(* CODESYS project tc3_cnc.library
   Company: Beckhoff Automation GmbH
   DefaultNamespace: Tc3_CNC
   Title: Tc3_CNC
   Description: TwinCAT CNC Library
   Placeholder: Tc3_CNC
   Author: Beckhoff Automation GmbH & Co. KG
   Version: 3.1.4000.18

Project tree, tasks and I/O mapping:
  libraries: Tc2_CncBase, * (Beckhoff Automation GmbH); Tc2_CncHli, * (Beckhoff Automation GmbH); Tc2_CncPlcopenP1, * (Beckhoff Automation GmbH); Tc2_EtherCAT, * (Beckhoff Automation GmbH); Tc2_Standard, * (Beckhoff Automation GmbH); Tc2_System, * (Beckhoff Automation GmbH); Tc2_Utilities, * (Beckhoff Automation GmbH); Tc3_Module, * (Beckhoff Automation GmbH)
  CNC/
    1 Init/
      program HLI3_Init [ST]
      function HLI3_SetAxisControlToPlc [ST]
      function HLI3_SetChannelControlToPlc [ST]
      function HLI3_UserInitialisation [ST]
    10 MessagesHandler/
      function CNCErrorDimensionToString [ST]
      function CNCErrorGetLogAxisId [ST]
      function CNCErrorMeaningToString [ST]
      function CNCErrorParameterToString [ST]
      function CNCErrorUnionToString [ST]
      function block FB_ChannelError [ST]
    11 Util/
      function F_GRAYCODE_TO_UINT [ST]
      function block FB_CNCWriteParameter [ST]
      function block FB_Uint_Udint [ST]
      function HLI3_FindAxisNameAndChannel [ST]
      function HLI3_FindHliAxisIdx [ST]
      function HLI3_GetEtherCATAxisInfo [ST]
      function block HLI3_SoftwareLimitSwitches [ST]
    12 CNC_Axis/
      function block FB_ActivateCompTable [ST]
      function block FB_CNCAxis [ST]
      function block FB_ReadSWLimitSwitches [ST]
      global variables GVL_CNC_AX
      function block HLI3_CNCAxis [ST]
      function block HLI3_CNCAxisBase [ST]: ACT_Init, ACT_Options, ACT_Parameter, ACT_PLCopen, ACT_Status
      data type ST_CNC_AX_Options
      data type ST_CNC_AX_Parameter
      data type ST_CNC_AX_PLCopen
      data type ST_CNC_AX_PLCopenStatus
      data type ST_CNC_AX_Status
    2 OperationMode/
      ModeManual/
        function HLI3_LogicalAxisInManualMode [ST]
        function block HLI3_ManualActivation [ST]
        function block HLI3_ManualExecution [ST]
        function block HLI3_ManualExecutionRapidMode [ST]
        function block HLI3_ManualModeHandler [ST]
        program PRG_AnalogJoystick [ST]
      function HLI3_AxisReset [ST]
      function HLI3_ChannelModeAuto [ST]
      function HLI3_ChannelModeManual [ST]
      function HLI3_ChannelModeMDI [ST]
      function HLI3_ChannelModeReference [ST]
      function HLI3_ChannelModeStandby [ST]
      function HLI3_ChannelReset [ST]
      function block HLI3_ChannelResetRequest [ST]
      function block HLI3_CNCChannel [ST]: AutoMDIStart, OpModes
      data type ST_CNC_CH_Options
    3 Control/
      function block FB_Diag [ST]
      function HLI3_ChannelSetBackwardMotion [ST]
      function HLI3_ChannelSetEmergencyStop [ST]
      function HLI3_ChannelSetFeedHold [ST]
      function HLI3_ChannelSetProgramBlockIgnore [ST]
      function HLI3_ChannelSetReducedFeed [ST]
      function HLI3_ChannelSetSingleBlock [ST]
      function HLI3_ChannelSetSuspendAxisOutput [ST]
      function HLI3_ClearReferencePosition [ST]
      function HLI3_GetActualAxisPos [ST]
      function HLI3_GetAxisReferenceState [ST]
      function block HLI3_GetChannelActiveG [ST]
      function HLI3_GetChannelError [ST]
      function block HLI3_GetChannelMessage [ST]
      function HLI3_GetChannelMode [ST]
      function HLI3_GetChannelState [ST]
      function HLI3_GetChannelStatusInfo [ST]
      function HLI3_GetFeedholdState [ST]
      function HLI3_GetIpoState [ST]
      function block HLI3_HandleSpindleTechno [ST]: A_HandleTechno, M_HandleTechnoAx, M_HandleTechnoCh, M_ManageAcknowledgement
      function block HLI3_HandleSpindleTechnoGearchange [ST]
      function HLI3_SetAxisGantryOn [ST]
      function HLI3_SetAxisOverride [ST]
      function HLI3_SetAxisReferenceCam [ST]
      function block HLI3_SetAxisReferenceOffset [ST]
      function HLI3_SetAxisReferencePosition [ST]
      function block HLI3_SetAxisRelease [ST]: AC_CanOpenDrive, AC_ClearError, AC_SercosDrive, AC_TerminalDrive
      function block HLI3_SetAxisSpindleStopAtProgramEnd [ST]
      function HLI3_SetAxisTrackingOperation [ST]
      function HLI3_SetChannelOverride [ST]
      function HLI3_SetChannelRapidOverride [ST]
      function HLI3_SetProbingSignal [ST]
    4 MHT-Function/
      function HLI3_ChannelResetHFunctions [ST]
      function HLI3_ChannelResetMFunctions [ST]
      function block HLI3_DoChannelHFunction [ST]
      function block HLI3_DoChannelMFunction [ST]
      function block HLI3_DoChannelTFunction [ST]
      function block HLI3_FastMFunctionHandler [ST]: ClearQueue, Dequeue, DequeuingRequired, Enqueue, RefreshQueue
      function block HLI3_FastMFunctionProvider [ST]
      function HLI3_QuitAxisMFunction [ST]
      function block HLI3_QuitChannelMHTFunction [ST]
    5 Variables/
      function block FB_ReadCNCVariables [ST]
      function HLI3_GetVEChannelBooleanValue [ST]
      function HLI3_GetVEChannelDIntValue [ST]
      function HLI3_GetVEChannelLRealValue [ST]
      function HLI3_GetVEChannelStringValue [ST]
      function HLI3_LinkVEChannelStructure [ST]
      function HLI3_SetVEChannelBooleanValue [ST]
      function HLI3_SetVEChannelDIntValue [ST]
      function HLI3_SetVEChannelLRealValue [ST]
      function HLI3_SetVEChannelStringValue [ST]
    6 BlockSearch/
      function block HLI3_BlockSearch [ST]
      function block ReadBlockCount [ST]
      function block ReadBlockNumber [ST]
      function block ReadBsAutoReturn [ST]
      function block ReadBsBlockCount [ST]
      function block ReadBsBlockNumber [ST]
      function block ReadBsCoveredDistance [ST]
      function block ReadBsDeviationMax [ST]
      function block ReadBsPass [ST]
      function block ReadBsType [ST]
      function block WriteBsAutoReturn [ST]
      function block WriteBsBlockCount [ST]
      function block WriteBsBlockNumber [ST]
      function block WriteBsCoveredDistance [ST]
      function block WriteBsDeviationMax [ST]
      function block WriteBsPass [ST]
      function block WriteBsType [ST]
    7 ToolManagement/
      program HLI3_ToolManagement [ST]: D_Command, T_Command, ToolLife_Command
    8 Mis/
      function block FB_WriteCNCZeroOffset [ST]
      function block FB_WriteCNCZeroOffsetDefault [ST]
      function block HLI_HandleMessages [ST]
      function block HLI_MoveSpindle [ST]
      function HLI3_CheckAxisValid [ST]
      function HLI3_CheckChannelValid [ST]
      program HLI3_CheckCNCAlive [ST]
      function HLI3_GetHliAxisIdx [ST]
      function HLI3_GetHliChannelIdx [ST]
      function HLI3_GetLogAxisId [ST]
      function HLI3_ResetSpindle [ST]
      function HLI3_SetPLCAlive [ST]
      program PB_10_CNC_Spindelkopplung [ST]
  DUTs/
    CNC_DataTyps/
      data type E_HLI_MM_KEYDIRECTION
      interface ITF_ToolAction: Commit, Tool
      data type ST_BlockSearch
      data type ST_ChannelSignals
      data type ST_CNC_TOOL_DATA_EXT
      data type ST_CNC_ToolChannel
      data type ST_CNCAxis
      data type ST_CncChannel
      data type ST_CncChannelInfo
      data type ST_CNCCmdModesStates
      data type ST_CNCG159VG
      data type ST_CncSystem
      data type ST_ManualMode
      data type ST_OpModes
      data type ST_OpStates
      data type ST_SyntaxCheck
      data type ST_TechnoAttributeData
      data type VEData
    CNC_FastMFunction/
      data type E_FastMFunctionState
      data type ST_FastMFunctionBufferItem
      data type ST_FastMFunctionData
      data type ST_FastMFunctionItem
    CNC_ManualMode/
      data type E_CNC_ManualType
      data type E_CNC_ManualZeroOffset
      data type ST_CNC_ManualOption
      data type ST_ManualModeAxis
      data type ST_ManualModeAxisKeys
      data type ST_ManualModeAxisParameter
      data type ST_ManualModeChannelParameter
      data type ST_ManualModeControlElements
      data type ST_ManualModeControlElementState
      data type ST_ManualModeJoystickParameter
      data type ST_ManualModeKeyHWUnit
      data type ST_ManualModeParameter
      data type ST_ManualModeState
    CNC_VariablesViewer/
      data type E_CNCVariablesType
      data type E_VEVariablesType
      data type ST_CNCVariablesViewer_Data
    CNC_WriteParameter/
      data type E_CNCParameterTypes
      data type ST_CNCParameter
    EventLogger/
      data type E_LogMethod
      data type ST_EventData
      data type ST_FileInfo
  GVLs/
    global variables Global_CNC
    global variables Global_CNCVariablesViewer
    global variables Global_ManualMode
  Version/
    global variables Global_Version
  Tc3_CNC.tmc
*)

// CNC/12 CNC_Axis/ST_CNC_AX_Options
TYPE ST_CNC_AX_Options :
STRUCT
	bResetCalibration	: BOOL;
	bReducedSpeed 		: BOOL;
	bReducedSpeedZone1  : BOOL;
	bReducedSpeedZone2  : BOOL;
	bProbingSignal		: BOOL;
	bActivateCompTable	: BOOL;	 
	strPathCompTable	: STRING(256);
END_STRUCT
END_TYPE

// CNC/12 CNC_Axis/ST_CNC_AX_Parameter
TYPE ST_CNC_AX_Parameter :
STRUCT
	nNumParameters 		: INT; 	
	bWriteParameter     : BOOL;	
	strTempPath			: STRING;
	ParamList			: ARRAY[0..199] OF ST_CNCParameter;
END_STRUCT
END_TYPE

// CNC/12 CNC_Axis/ST_CNC_AX_PLCopen
TYPE ST_CNC_AX_PLCopen :
STRUCT	
	nOverride 		     : UINT; 		// [ 0.1% ]
	bExecuteHoming		 : BOOL;
	bCamSignal			 : BOOL;
	bExecuteMoveAbsolute : BOOL;
 	bExecuteStop 		 : BOOL;
	bExecuteReset 		 : BOOL;	
	fPosition 			 : LREAL;      // [ mm or degree ]
	fVelocity       	 : LREAL;      // [ mm/min or degree/min ]
	fAcceleration   	 : LREAL;	  // [ mm/s^2 or degree/s^2 ]
	fJerk   			 : LREAL;	  // [ mm/s^3 or degree/s^3 ]
END_STRUCT
END_TYPE

// CNC/12 CNC_Axis/ST_CNC_AX_PLCopenStatus
TYPE ST_CNC_AX_PLCopenStatus :
STRUCT	
	bError 				: BOOL;
	nErrorID 			: DINT;
	bMoveAbsoluteDone 	: BOOL;
	bHomingDone 		: BOOL;
	bStopDone 			: BOOL;
	bResetDone 			: BOOL;
END_STRUCT
END_TYPE

// CNC/12 CNC_Axis/ST_CNC_AX_Status
TYPE ST_CNC_AX_Status :
STRUCT
	bHomingDone 	: BOOL;
	fSetPosACS		: LREAL;	// [ mm or degree ] 
	fActPosACS		: LREAL;	// [ mm or degree] 
	fActVelo		: LREAL;	// [ mm or degree or rpm ]
	nCNCErrorID 	: UDINT;	// CNC Axis Error Id
	PLCopen   		: ST_CNC_AX_PLCopenStatus;
END_STRUCT
END_TYPE

// CNC/2 OperationMode/ST_CNC_CH_Options
TYPE ST_CNC_CH_Options :
STRUCT
	bReferenceModeStartRequired : BOOL;
END_STRUCT
END_TYPE

// DUTs/CNC_DataTyps/E_HLI_MM_KEYDIRECTION
TYPE E_HLI_MM_KEYDIRECTION :
(
	KEY_DIR_NEGATIVE := -1,
	KEY_DIR_NOT_PRESSED := 0,
	KEY_DIR_POSITIVE := 1
);
END_TYPE

// DUTs/CNC_DataTyps/ST_BlockSearch
TYPE ST_BlockSearch :
STRUCT
	/// Block Search 
	Active: BOOL;
	/// Edge signal 
	bStartRead: BOOL;
	/// Edge signal 
	bStartWrite: BOOL;
	/// 0 - no block search
	///                                    3 - start position by block count
	///                                    4 - start position by block nr
	///                                    5 - start position BY individual mark 
	nType: UINT;
	fDistance: LREAL;
	bAutoReturn: BOOL;
	nDeviationMax: UDINT;
	nBlockNumber: DINT;
	nPass: DINT;
	nBlockCount: DINT;
END_STRUCT
END_TYPE

// DUTs/CNC_DataTyps/ST_ChannelSignals
TYPE ST_ChannelSignals :
STRUCT
	DoSingleBlock: BOOL;
	SingleBlock: BOOL;
	FeedHold: BOOL;
	Backward: BOOL;
	PrgBlockIgnore: BOOL;
	M01Stop: BOOL;
END_STRUCT
END_TYPE

// DUTs/CNC_DataTyps/ST_CNC_TOOL_DATA_EXT
TYPE ST_CNC_TOOL_DATA_EXT :
STRUCT
	tool_desc: CNC_TOOL_DESC;
	tool_life: CNC_TOOL_LIFE_DATA;
	dist_max: LREAL;
	time_max: LREAL;
	/// 0.1 µm 
	laenge: DINT;
	/// 0.1 µm 
	laenge_delta: DINT;
	/// 0.1 µm 
	radius: DINT;
	/// 0.1 µm 
	radius_delta: DINT;
	/// position in tool holder 
	pos: DINT;
	/// 0.1 µm 
	tolerancePos: DINT;
	/// 0.1 µm 
	toleranceNeg: DINT;
END_STRUCT
END_TYPE

// DUTs/CNC_DataTyps/ST_CNC_ToolChannel
TYPE ST_CNC_ToolChannel :
STRUCT
	
	bToolRequest: 			BOOL;   (* rising edge starts request of tool data from HMI, HMI resets to false after reading *)
	nToolRequestID: 		DINT;   (* tool id for request *)
	nToolRequestIDSister:	DINT;	(* tool sister id for request, 0 if not needed *)
	nToolRequestIDVariant:	DINT;   (* tool variant id for request, 0 if not needed *)		
	
	bToolRequestPrepData:	BOOL;   (* rising edge starts request of tool data to structure stPrepTool *)
	nToolRequestPrepId: 	DINT;   (* tool id for pepRequest *)
	
	bOldToolDataExist:		BOOL;   (* rising edge commands the HMI to read oldData from stOldTool *)
		
	stActTool:	 			ST_CNC_TOOL_DATA_EXT; (* complete tool data for actual tool that will be transfered FROM HMI  *)
	stOldTool:	 			ST_CNC_TOOL_DATA_EXT; (* complete tool data for odlTool that will be transfered TO HMI *)
	stPrepTool:				ST_CNC_TOOL_DATA_EXT; (* complete tool data for preTool that will be transfered FROM HMI *)
	
	stActT:					ST_CNC_TOOL_DATA_EXT; (* (internal) tool data for the actual requested T *)
	
	nToolInCnc:				DINT;	(* main tool id of tool actually in cnc *)
	nToolInCncSister: 		DINT;	(* sister tool id of tool actually in cnc *)
	nToolInCncVariant:		DINT;	(* variant tool id of tool actually in cnc *)
	
	bResetToolRequest:		BOOL;
	
	TCommand:				ITF_ToolAction;  (* the method Commit is called before data for T is transfered to CNC. The process os stopped until the commit method returns true *)
	DCommand:				ITF_ToolAction;  (* the method Commit is called before data for D is transfered to CNC. The process os stopped until the commit method returns true *)
	ToolLifeCommand:		ITF_ToolAction;  (* the method Commit is called before data for ToolLife is transfered to HMI. The process os stopped until the commit method returns true *)	

END_STRUCT
END_TYPE

// DUTs/CNC_DataTyps/ST_CNCAxis
TYPE ST_CNCAxis :
STRUCT
	nHliAxisIdx : INT := -1;
    strLogName	: STRING(HLI_ACHS_NAME_LAENGE);
	{attribute 'hide'}
	nCNCErrorID : UDINT;	
END_STRUCT
END_TYPE

// DUTs/CNC_DataTyps/ST_CncChannel
TYPE ST_CncChannel :
STRUCT
	nLogNumber  : DINT := -1;
    strLogName	: STRING(HLI_ACHS_NAME_LAENGE);
	/// Operation Mode 
	Mode: ST_OpModes;
	/// Operation States 
	State: ST_OpStates;
	/// Selected Mode 
	ActMode: UDINT;
	/// Selected Mode as string 
	ActModeString: STRING;
	/// Selected State 
	ActState: UDINT;
	/// Selected State as string 
	ActStateString: STRING;
	/// Block Search : Act. Distance 
	ActDistance: LREAL;
	/// Block Search : Act. Block Count 
	ActBlockCount: UDINT;
	actM_r: STRING(5);
	actH_r: STRING(5);
	/// M-Functions 
	M: ARRAY[0..999] OF ST_TechnoAttributeData;
	/// H-Functions 
	H: ARRAY[0..999] OF ST_TechnoAttributeData;	
	/// Fehlerflag des Kanals 
	Error: BOOL;	
	/// Message from NC program to PLC 
	Message: STRING(HLI_MSG_CONTENT_STRL);
	// Data for tool handling
	ToolData      :  ST_CNC_ToolChannel;
	
END_STRUCT
END_TYPE

// DUTs/CNC_DataTyps/ST_CncChannelInfo
TYPE ST_CncChannelInfo :
STRUCT
	nHliChannelIdx : INT := -1;
    strLogName	: STRING(HLI_CHANNEL_NAME_LAENGE);
END_STRUCT
END_TYPE

// DUTs/CNC_DataTyps/ST_CNCCmdModesStates
TYPE ST_CNCCmdModesStates :
	STRUCT	
	stModes : ST_OpModes;
	stStates : ST_OpStates;
	END_STRUCT
END_TYPE

// DUTs/CNC_DataTyps/ST_CNCG159VG
TYPE ST_CNCG159VG :
STRUCT
	sTarget: STRING(95);
	dValue: DINT;
END_STRUCT
END_TYPE

// DUTs/CNC_DataTyps/ST_CncSystem
TYPE ST_CncSystem :
STRUCT
	/// Initialization of HLI done 
	bHLIInit: BOOL;
	/// Initialization of PLCopenPlatform done 
	bPLCopenPlatformInit : BOOL;
	/// Initialization of user data done
	bUserInitDone: BOOL;
	/// Error init HLI-Interfaces 
	bInitError: BOOL;
	/// ErrorId during init HLI-Interfaces 
	nInitErrorId: UDINT;
	Channel: ARRAY[0..HLI_SYS_CH_MAXIDX] OF ST_CncChannel;
    LogAxisNo : ARRAY[0..MAX_SYS_LOG_AXIS_INDEX] OF ST_CncAxis;	
	LogChannelNo : ARRAY[0..HLI_SYS_CH_MAXIDX] OF ST_CncChannelInfo;    	
END_STRUCT
END_TYPE

// DUTs/CNC_DataTyps/ST_ManualMode
TYPE ST_ManualMode :
STRUCT
	bKeyPos: BOOL;
	bKeyNeg: BOOL;
	bKeyRapid: BOOL;
	nLogAxisNumber: UINT;
	nInc: UDINT;
	nManualTyp: UINT;
	stManualOption			: ST_CNC_ManualOption;
	nSpeed: UINT;
	/// Handradauflösung in 0.1 um / Umdrehung 
	nHwResolution: UDINT;
END_STRUCT
END_TYPE

// DUTs/CNC_DataTyps/ST_OpModes
TYPE ST_OpModes :
STRUCT
	Standby: BOOL;
	Auto: BOOL;
	Manual: BOOL;
	MDI: BOOL;	
	Homing: BOOL;
END_STRUCT
END_TYPE

// DUTs/CNC_DataTyps/ST_OpStates
TYPE ST_OpStates :
STRUCT
	Selected: BOOL;
	Ready: BOOL;
	Active: BOOL;
	Hold: BOOL;
	Reset: BOOL;
END_STRUCT
END_TYPE

// DUTs/CNC_DataTyps/ST_SyntaxCheck
TYPE ST_SyntaxCheck :
STRUCT
	/// SyntaxCheck 
	nType: INT;
END_STRUCT
END_TYPE

// DUTs/CNC_DataTyps/ST_TechnoAttributeData
TYPE ST_TechnoAttributeData :
STRUCT
	bState_rw: BOOL;
	nFunctionNumber_r: UDINT;
	nTime_r: DINT;
	nBlockNumber_r: UDINT;
	nPrgLineNumber_r: UDINT;
	nArgument_r: DINT;
	{attribute 'hide'}
	bRes: BOOL;
END_STRUCT
END_TYPE

// DUTs/CNC_DataTyps/VEData
TYPE VEData :
STRUCT
	AHLI_UNS32_Data: ARRAY[0..HLI_EXT_VAR32_MAXIDX] OF UDINT;
END_STRUCT
END_TYPE

// DUTs/CNC_FastMFunction/E_FastMFunctionState
(****************************************************************************************)
(* POU:		E_FastMFunctionState                     									*)
(* Type:	ENUM																		*)
(* Author: 	RCH		                                             						*)
(* Date: 	14/10/29																	*)
(* Rev.: 	1.0                                               							*)
(* ------------------------------------------------------------------------------------ *)
(* Desc.:	Defines the state of an digital output handled by instances of FB			*)
(*			HLI3_FastMFunctionHandler.													*)
(* ------------------------------------------------------------------------------------ *)
(* Rev.:	<Enter revision number here>												*)
(* Date:	<Enter revision data here>				                                   	*)
(* Author:	<Enter author´s shortcut here>											 	*)
(* Desc.:	<Enter description here>													*)
(****************************************************************************************)
TYPE E_FastMFunctionState :
(
	EMPTY	:= 0,	(* Not switched yet *)
	OFF 	:= 1,	(* Switched OFF *)
	ON 		:= 2	(* Switched ON *)
);
END_TYPE

// DUTs/CNC_FastMFunction/ST_FastMFunctionBufferItem
(****************************************************************************************)
(* POU:		ST_FastMFunctionBufferItem                     								*)
(* Type:	STRUCT																		*)
(* Author: 	RCH		                                             						*)
(* Date: 	14/10/29																	*)
(* Rev.: 	1.0                                               							*)
(* ------------------------------------------------------------------------------------ *)
(* Desc.:	Defines data content for a single fast M function switch event managed 		*)
(*			internally by instances of HLI3_FastMFunctionHandler.						*) 
(* ------------------------------------------------------------------------------------ *)
(* Rev.:	<Enter revision number here>												*)
(* Date:	<Enter revision data here>				                                   	*)
(* Author:	<Enter author´s shortcut here>											 	*)
(* Desc.:	<Enter description here>													*)
(****************************************************************************************)
TYPE ST_FastMFunctionBufferItem :
STRUCT
	eState			: E_FastMFunctionState;		(* The target switch state *)
	nSwitchTime		: DINT;						(* The calculated switch time *)
END_STRUCT
END_TYPE

// DUTs/CNC_FastMFunction/ST_FastMFunctionData
(****************************************************************************************)
(* POU:		ST_FastMFunctionData                     								*)
(* Type:	STRUCT																		*)
(* Author: 	RCH		                                             						*)
(* Date: 	14/10/29																	*)
(* Rev.: 	1.0                                               							*)
(* ------------------------------------------------------------------------------------ *)
(* Desc.:	Defines preprocessed information about MOS_TS M functions and their			*)
(*			metadata generated by HLI3_FastMFunctionProvider and consumed by 			*)
(*			HLI3_FastMFunctionHandler(s)												*) 
(* ------------------------------------------------------------------------------------ *)
(* Rev.:	<Enter revision number here>												*)
(* Date:	<Enter revision data here>				                                   	*)
(* Author:	<Enter author´s shortcut here>											 	*)
(* Desc.:	<Enter description here>													*)
(****************************************************************************************)
TYPE ST_FastMFunctionData :
STRUCT
	bCycleTimeExceeded	: BOOL;																	(* TRUE if the cycle time has been exceeded and therefore the data is unvalid *)
	bDataValid			: BOOL;																	(* TRUE if data is valid *)
	nFunctionCount		: UINT;																	(* Number of M function data sets contained in 'astItem' *)
	astItem				: ARRAY[0..MAX_FAST_M_FUNC_ITEM_IDX] OF ST_FastMFunctionItem;			(* M function metadata items *)
END_STRUCT
END_TYPE

// DUTs/CNC_FastMFunction/ST_FastMFunctionItem
(****************************************************************************************)
(* POU:		ST_FastMFunctionItem                     									*)
(* Type:	STRUCT																		*)
(* Author: 	RCH		                                             						*)
(* Date: 	14/10/29																	*)
(* Rev.: 	1.0                                               							*)
(* ------------------------------------------------------------------------------------ *)
(* Desc.:	Defines M function metadata content provided by HLI3_FastMFunctionProvider	*)
(* ------------------------------------------------------------------------------------ *)
(* Rev.:	<Enter revision number here>												*)
(* Date:	<Enter revision data here>				                                   	*)
(* Author:	<Enter author´s shortcut here>											 	*)
(* Desc.:	<Enter description here>													*)
(****************************************************************************************)
TYPE ST_FastMFunctionItem :
STRUCT
	nFunctionNo		: UINT;			(* M function number *)
	nOffset			: DINT;			(* Time offset with respect to the block change time *)
	nCycleCount		: UDINT;		(* PLC cycle counter *)
END_STRUCT
END_TYPE

// DUTs/CNC_ManualMode/E_CNC_ManualType
TYPE E_CNC_ManualType :
(
	NoManualMode := 0,
	Handwheel := 1,
	TippMode := 2,
	JogMode := 3,
	JoystickMode := 4,
	DigitalJoystick := 5
);
END_TYPE

// DUTs/CNC_ManualMode/E_CNC_ManualZeroOffset
TYPE E_CNC_ManualZeroOffset :
(
	G53 := 0,
	G54 := 1,
	G55 := 2,
	G56 := 3,
	G57 := 4,
	G58 := 5,
	G59 := 6
);
END_TYPE

// DUTs/CNC_ManualMode/ST_CNC_ManualOption
TYPE ST_CNC_ManualOption :
STRUCT
	bTrafoActive: BOOL;
	bEcsActive: BOOL;
	bCAXActive: BOOL;
	eZeroOffset: E_CNC_ManualZeroOffset;
END_STRUCT
END_TYPE

// DUTs/CNC_ManualMode/ST_ManualModeAxis
TYPE ST_ManualModeAxis :
STRUCT
	nLogAxisNr: UINT;
	nSpeed: UDINT;
END_STRUCT
END_TYPE

// DUTs/CNC_ManualMode/ST_ManualModeAxisKeys
TYPE ST_ManualModeAxisKeys :
STRUCT
	/// static signal + 
	bKeyPos: BOOL;
	/// static signal - 
	bKeyNeg: BOOL;
	/// static signal Rapid 
	bKeyRapid: BOOL;
END_STRUCT
END_TYPE

// DUTs/CNC_ManualMode/ST_ManualModeAxisParameter
TYPE ST_ManualModeAxisParameter :
STRUCT
	stControlUnit: ARRAY[0..HLI_KEY_MAXIDX] OF ST_ManualModeAxis;
END_STRUCT
END_TYPE

// DUTs/CNC_ManualMode/ST_ManualModeChannelParameter
TYPE ST_ManualModeChannelParameter :
STRUCT
	/// Number of channel 
	nChanIdx: INT := -1;
	nInc: UDINT;
	/// Aufloesung des Achsverfahrwegs bei einer Handradumdrehung Einheit: 0.1um / Handradumdrehung
	nHandwheelResolution: DINT;	 	
	/// configuration 
	eManualType: E_CNC_ManualType;
	stManualOption: ST_CNC_ManualOption;
	strInitParameter: STRING;
END_STRUCT
END_TYPE

// DUTs/CNC_ManualMode/ST_ManualModeControlElements
TYPE ST_ManualModeControlElements :
STRUCT
	stControlKeys: ARRAY[0..HLI_KEY_MAXIDX] OF ST_ManualModeAxisKeys;
	stControlJoystickValue: ARRAY[0..HLI_KEY_MAXIDX] OF DINT;
	/// Es können 6 Handräder verwendet werden 
	nHandwheelInc: ARRAY[0..HLI_HW_MAXIDX] OF DINT;
END_STRUCT
END_TYPE

// DUTs/CNC_ManualMode/ST_ManualModeControlElementState
TYPE ST_ManualModeControlElementState :
STRUCT
	stKeyUnit: ARRAY[0..HLI_KEY_MAXIDX] OF ST_ManualModeKeyHWUnit;
	stHWUnit: ARRAY[0..HLI_HW_MAXIDX] OF ST_ManualModeKeyHWUnit;
END_STRUCT
END_TYPE

// DUTs/CNC_ManualMode/ST_ManualModeJoystickParameter
TYPE ST_ManualModeJoystickParameter :
STRUCT
	/// static signal : Analog Min Value 
	AnalogValueMin: DINT;
	/// static signal : Analog Max Value 
	AnalogValueMax: DINT;
	/// Dead Band for Zero Value 
	AnalogValueZeroDeadBand: DINT;
END_STRUCT
END_TYPE

// DUTs/CNC_ManualMode/ST_ManualModeKeyHWUnit
TYPE ST_ManualModeKeyHWUnit :
STRUCT
	nLogAxisId: UINT;
	nChan: INT := -1;
	nInputParameterIdx: INT;
END_STRUCT
END_TYPE

// DUTs/CNC_ManualMode/ST_ManualModeParameter
TYPE ST_ManualModeParameter :
STRUCT
	stAxisParameter: ST_ManualModeAxisParameter;
	stJoystickParameter: ST_ManualModeJoystickParameter;
	stChannelParameter: ST_ManualModeChannelParameter;	
END_STRUCT
END_TYPE

// DUTs/CNC_ManualMode/ST_ManualModeState
TYPE ST_ManualModeState :
STRUCT
	arrAxisInG201: ARRAY[0..HLI_KEY_MAXIDX] OF UINT;
END_STRUCT
END_TYPE

// DUTs/CNC_VariablesViewer/E_CNCVariablesType
{attribute 'qualified_only'}
{attribute 'strict'}
TYPE E_CNCVariablesType :
(
	none :=0,
	VE,
    P,
    VP,
    VS,
    VL        
);
END_TYPE

// DUTs/CNC_VariablesViewer/E_VEVariablesType
{attribute 'qualified_only'}
{attribute 'strict'}
TYPE E_VEVariablesType :
(
	none := 0,
	BOOLEAN,
	SGN08,
	UNS08,
	SGN16,
	UNS16,
	SGN32,
	UNS32,
	REAL64,
	VESTRING	
);
END_TYPE

// DUTs/CNC_VariablesViewer/ST_CNCVariablesViewer_Data
TYPE ST_CNCVariablesViewer_Data :
STRUCT
	strName : STRING;
	strValue  : STRING(799);
END_STRUCT
END_TYPE

// DUTs/CNC_WriteParameter/E_CNCParameterTypes
TYPE E_CNCParameterTypes :
(
	CNC_ChannelParameter := 10,
	CNC_AxisParameter := 11,
	CNC_ZeroOffsets := 12,
	CNC_ToolParameter := 13,
	CNC_ClampPosition := 14
);
END_TYPE

// DUTs/CNC_WriteParameter/ST_CNCParameter
TYPE ST_CNCParameter :
STRUCT
	strName: STRING;
	strValue: STRING;
	strDescription: STRING;
END_STRUCT
END_TYPE

// DUTs/EventLogger/E_LogMethod
TYPE E_LogMethod :
(
	Static := 0,
	RisingTrig := 1,
	FallingTrig := 2
);
END_TYPE

// DUTs/EventLogger/ST_EventData
TYPE ST_EventData :
STRUCT
	nParam1: DINT;
	nParam2: STRING;	
END_STRUCT
END_TYPE

// DUTs/EventLogger/ST_FileInfo
TYPE ST_FileInfo :
STRUCT
	nSource: UDINT;
	nOffset: UDINT;
	sFilename: STRING(260);
END_STRUCT
END_TYPE

// CNC/12 CNC_Axis/GVL_CNC_AX
VAR_GLOBAL
	fbCNC_AX_WriteParameter			: FB_CNCWriteParameter;	
	bCNC_AX_WriteParameterLock 		: BOOL;
	fbActivateCompTable 			: FB_ActivateCompTable;
	bCNC_AX_ActivateCompTableLock  	: BOOL;
END_VAR

// GVLs/Global_CNC
VAR_GLOBAL
	CNCSystem						: ST_CncSystem;
END_VAR

(****************************************************************************************)
(*	  	Global constants used by the fast M function handling process (MOS_TS)			*)
(****************************************************************************************)
VAR_GLOBAL CONSTANT
	MAX_FAST_M_FUNC_ITEM_IDX	: UINT	:= 7;			(* Max. index of fast M functions processed by HLI3_FastMFunctionProvider per PLC cycle *) 
	MAX_FAST_M_FUNC_QUEUE_IDX	: UINT	:= 63;			(* Max. index of fast M function switch events buffered by HLI3_FastMFunctionHandler *) 
	MAX_FAST_M_FUNC_OUTPUT_IDX	: UINT	:= 124;			(* Max. index of fast M function oversampling output byte array *)			
	MAX_SYS_LOG_AXIS_INDEX		: UINT  := 255;			(* Max. Index of Log. Axis Id *) 				
END_VAR

// GVLs/Global_CNCVariablesViewer
{attribute 'pack_mode' := '1'}
VAR_GLOBAL
	stCNCVariablesViewer_Data : ARRAY[0..MAX_CNC_VAR_LIST_IDX] OF ST_CNCVariablesViewer_Data;
	eVariablesType : E_CNCVariablesType;

END_VAR

VAR_GLOBAL CONSTANT
	MAX_CNC_VAR_LIST_IDX : UINT := 200;
END_VAR

// GVLs/Global_ManualMode
VAR_GLOBAL
	/// Manual mode control structures 
	stManualModeParameter: ARRAY[0..HLI_SYS_CH_MAXIDX] OF ST_ManualModeParameter;
	stManualModeControlElements: ARRAY[0..HLI_SYS_CH_MAXIDX] OF ST_ManualModeControlElements;
	stManualModeState: ARRAY[0..HLI_SYS_CH_MAXIDX] OF ST_ManualModeState;
	stManualModeControlElementState : ST_ManualModeControlElementState;
END_VAR

// Version/Global_Version
{attribute 'TcGenerated'}
// This function has been automatically generated from the project information.
VAR_GLOBAL CONSTANT
	{attribute 'const_non_replaced'}
	{attribute 'linkalways'}
	stLibVersion_Tc3_CNC : ST_LibVersion := (iMajor := 3, iMinor := 1, iBuild := 4000, iRevision := 18, sVersion := '3.1.4000.18');
END_VAR

// CNC/1 Init/HLI3_Init
PROGRAM HLI3_Init
VAR
	Hli: MCV_HliInterface;
	bFirstCycle: BOOL := TRUE;
	ipSrv: ITComObjectServer;
	oidCnc: UDINT := 16#5500001;
	bUnregister: BOOL;
	MessageOutput: R_TRIG;
	nHliAxisIdx	: INT;
	nHliChannelIdx: INT;
	
	PlatformBase: MCV_PlatformBase;
	P1_Platform: MCV_P1_Platform;
END_VAR

(* ========================================================= *)
(*    PRG: HLI_Init                                          *)
(* --------------------------------------------------------- *)
(*   Desc:                                                   *)
(* Author: MK                                                *)
(*   Date: 21.12.2011                                        *)
(*   Rev.: 1.0                                               *)
(*   Date: 06.08.2013                                        *)
(*   Rev.: 1.1 TV   Error Message if HLI not initialized	 *)
(*   Date: 05.01.2017                                        *)
(*   Rev.: 1.2 TV   BugFix Init LogAxisNo Array              *)
(*   Date: 06.06.2017                                        *)
(*   Rev.: 1.3 TV  new LogChannelNo            	 			 *)
(*   Date: 08.11.2017                                        *)
(*   Rev.: 1.4 TV  new FB call fbCNC_AX_WriteParameter       *)
(*   			   new FB call 	fbActivateCompTable       	 *)
(* ========================================================= *)



IF bFirstCycle THEN
	Hli();					(* initialize HLI *)
	bFirstCycle := FALSE;
END_IF


IF Hli.Initialized  = TRUE
THEN
	(* User initialization, used during start of PLC once *)
	IF CncSystem.bUserInitDone = FALSE THEN
		(* Initialisierungen auf dem HLI-Interface *)
		CncSystem.bUserInitDone := HLI3_UserInitialisation();
		//ADSLOG(strMsg:='High Level Interfaces initialized: %s', nDINT:=0, strArg:='');
	END_IF

	IF (NOT CNCSystem.bHLIInit) THEN
		FOR nHliAxisIdx := 0 TO UDINT_TO_INT(gNrAx-1) DO
        	IF HLI3_CheckAxisValid(nHliAxisIdx) THEN
            	CNCSystem.LogAxisNo[gpAx[nHliAxisIdx]^.head.log_ax_nr_r].nHliAxisIdx := nHliAxisIdx;
                CNCSystem.LogAxisNo[gpAx[nHliAxisIdx]^.head.log_ax_nr_r].strLogName   := gpAx[nHliAxisIdx]^.lr_state.log_name_r.zeichen;                                 
           	END_IF
		END_FOR
		
		FOR nHliChannelIdx := 0 TO UDINT_TO_INT(gNrCh-1) DO
        	IF HLI3_CheckCHannelValid(nHliChannelIdx) THEN
				CNCSystem.Channel[nHliChannelIdx].nLogNumber := gpCh[nHliChannelIdx]^.head.channel_nr;
				CNCSystem.Channel[nHliChannelIdx].strLogName := gpCh[nHliChannelIdx]^.head.channel_name_r.zeichen; 
            	CNCSystem.LogChannelNo[gpCh[nHliChannelIdx]^.head.channel_nr].nHliChannelIdx := nHliChannelIdx;
            	CNCSystem.LogChannelNo[gpCh[nHliChannelIdx]^.head.channel_nr].strLogName := gpCh[nHliChannelIdx]^.head.channel_name_r.zeichen;				                                                 
           	END_IF
		END_FOR
		
	END_IF
	
	(* initialization finished *)
	CNCSystem.bHLIInit := TRUE;
	
	(* call tool management *)
	HLI3_ToolManagement();
	
	// Global FB to Write Axis Parameters to the CNC
	fbCNC_AX_WriteParameter();		
	// Global FB to Activate Compensation Table 
	fbActivateCompTable();
	
	PlatformBase();

	CNCSystem.bPLCopenPlatformInit := PlatformBase.Done; 
	
	IF CNCSystem.bPLCopenPlatformInit THEN
		P1_Platform();
	END_IF

ELSE
	MessageOutput(CLK:=Hli.Error);
	IF Hli.Error = TRUE	THEN
		(* High Level Interface (HLI) not initialized *)
		IF MessageOutput.Q THEN
			ADSLOGDINT(	msgCtrlMask := ADSLOG_MSGTYPE_ERROR OR
												ADSLOG_MSGTYPE_MSGBOX OR
												ADSLOG_MSGTYPE_LOG,
							msgFmtStr := 'High Level Interface (HLI) not initialized! Errorcode: %d',
							dintArg := Hli.ErrorID);
		END_IF
		CNCSystem.nInitErrorId := Hli.ErrorID;
		CNCSystem.bInitError := TRUE;
	END_IF;	
END_IF

END_PROGRAM

// CNC/1 Init/HLI3_UserInitialisation
FUNCTION HLI3_UserInitialisation : BOOL
VAR
	idx: UDINT;
END_VAR

(* ========================================================= *)
(*    FUN: HLI_UserInitialisation                            *)
(* --------------------------------------------------------- *)
(*   Desc:                                                   *)
(* Author: MK                                                *)
(*   Date: 18.07.2002                                        *)
(*   Rev.: 1.0 												 *)
(*         1.1 MiB 19.12.2012 Tc3 Anpassung                  *)
(*         1.2 TV 30.06.2015  Function call SetChannelControl*)
(*							  in a For Loop					 *)											  							  
(* ========================================================= *)

(* please do reset the plc program, if you change something in this module
	or in modules are in the sublevel *)

(* Axis Control *)	
HLI3_SetAxisControlToPlc();	
	
FOR idx := 0 TO gNrch - 1 DO
	HLI3_SetChannelControlToPlc(nChan:=UDINT_TO_INT(idx));
END_FOR

HLI3_UserInitialisation := TRUE;

END_FUNCTION

// CNC/1 Init/HLI3_SetAxisControlToPlc
FUNCTION HLI3_SetAxisControlToPlc : BOOL
VAR
	idx: UDINT;
END_VAR

(* ========================================================= *)
(*    FUN: HLI3_SetAxisControlToPlc                          *)
(* --------------------------------------------------------- *)
(*   Desc:                                                   *)
(*   Author: MiB                                             *)
(*   Date: 19.11.2012                                        *)
(*   Rev.: 1.0                                               *)
(* ========================================================= *)

(* control to the plc *)
FOR idx := 0 TO gNrAx - 1 DO

	IF (idx < INT_TO_UDINT(HLI_SYS_AX_MAX)) THEN 
		IF gpAx[idx] <> 0 THEN						// check for zero pointer
			// PLC_Present for all axis
			gpAx[idx]^.head.plc_present_w 								:= TRUE;
		
			(* declare axis for reference *)
			gpAx[idx]^.lr_mc_control.reference_cam.enable_w 			:= TRUE;
	
			(* enable signals for real drives *)
			gpAx[idx]^.lr_mc_control.torque_permission.enable_w			:= TRUE;
			gpAx[idx]^.lr_mc_control.release_feedhold.enable_w 			:= TRUE;
			gpAx[idx]^.lr_mc_control.drive_on.enable_w 					:= TRUE;
			
			(* set reference postion offset *)
			gpAx[idx]^.lr_mc_control.set_reference_position.enable_w	:= TRUE;
			gpAx[idx]^.lr_mc_control.refpos_position.enable_w			:= TRUE;
			gpAx[idx]^.lr_mc_control.reference_cam.enable_w				:= TRUE;
			
			(* enable external commanding of an axis *)
			gpAx[idx]^.lr_mc_control.add_cmd_values.enable_w 			:= TRUE;
	
			(* enable the axis to tracking operation (follow up) *)
			gpAx[idx]^.lr_mc_control.follow_up.enable_w 				:= TRUE;
		END_IF
	END_IF
END_FOR

HLI3_SetAxisControlToPlc												:= TRUE;

END_FUNCTION

// CNC/1 Init/HLI3_SetChannelControlToPlc
FUNCTION HLI3_SetChannelControlToPlc : BOOL
VAR_INPUT
	nChan: INT;
END_VAR

(* ========================================================= *)
(*    FUN: HLI3_SetChannelControlToPlc                       *)
(* --------------------------------------------------------- *)
(*   Desc:                                                   *)
(* Author: MK                                                *)
(*   Date: 18.07.2002                                        *)
(*   Rev.: 1.0                                               *)
(*   Date: 19.11.2012                                        *)
(*   Rev.: 1.1 MiB TC3 0 based index                         *)
(* ========================================================= *)


IF (NOT HLI3_CheckChannelValid(nChannel := nCHan)) THEN
	HLI3_SetChannelControlToPlc											:= FALSE;
	RETURN; (* A b b r u c h *)
END_IF


(* PLC_Present for the channel *)
gpCh[nChan]^.head.plc_present_w 									:= TRUE;

(* reset *)
gpCh[nChan]^.bahn_lc_control.plc_reset.enable_w 					:= TRUE;
gpCh[nChan]^.channel_mc_control.mode_and_state.enable_w				:= TRUE;

(* override *)
gpCh[nChan]^.bahn_mc_control.override_feedrate.enable_w 			:= TRUE;

(* FeedHold *)
gpCh[nChan]^.bahn_mc_control.feedhold.enable_w 					:= TRUE;

(* Single Step *)
gpCh[nChan]^.bahn_mc_control.single_block.enable_w 				:= TRUE;

(* BackwardMotion *)
gpCh[nChan]^.bahn_mc_control.backward_motion.enable_w 			:= TRUE;

(* ReducedFeed *)
gpCh[nChan]^.bahn_mc_control.reduced_speed.enable_w 				:= TRUE;

(* Handwheel *)
gpCh[nChan]^.hb_mc_control.handwheel_incs[0].enable_w 			:= TRUE;

(* Channel switch "jog of path" *)
gpCh[nChan]^.bahn_mc_control.suspend_axis_output.enable_w 		:= TRUE;

(* logon for error messages *)
gpCh[nChan]^.mc_error.enable_w 									:= TRUE;

(* program block ignore *)
gpCh[nChan]^.decoder_mc_control.program_block_ignore.enable_w	:= TRUE;

(* Syntax Check *)
gpCh[nChan]^.decoder_mc_control.execution_mode.enable_w			:= TRUE;

(* Optional stop M01 *)
gpCh[nChan]^.bahn_mc_control.m01_stop_enable.enable_w			:= TRUE;

(* Emergency Stop *)
gpCh[nChan]^.bahn_mc_control.emergency_stop.enable_w				:= TRUE;

HLI3_SetChannelControlToPlc 												:= TRUE;

END_FUNCTION

// CNC/8 Mis/HLI3_CheckChannelValid
FUNCTION HLI3_CheckChannelValid : BOOL
VAR_INPUT
	nChannel: INT;
END_VAR

(* ========================================================= *)
(*    FUN: HLI3_CheckChannelValid                            *)
(* --------------------------------------------------------- *)
(*   Desc: Check if channel ID is valid for HLI access       *)
(*   Author: MiB                                             *)
(*   Date: 19.11.2012                                        *)
(*   Last: 21.06.2013										 *)
(*   Rev.: 1.1                                               *)
(* --------------------------------------------------------- *)
(*   Desc: Corrected IF statement (line 14)		 	      	 *)
(*   Author: RCH                                             *)
(*   Date: 16.09.2013                                        *)
(*   Rev.: 1.2                                               *)
(* ========================================================= *)

IF (nChannel < 0) THEN
	HLI3_CheckChannelValid:= FALSE;
	RETURN; (* A b b r u c h *)
ELSIF (nChannel >=  UDINT_TO_INT(gNrCh) ) OR		(* check for channel no *)
       (gpCh[nChannel] = 0) 				  (* check for zero pointer *)
THEN
	HLI3_CheckChannelValid:= FALSE;
	RETURN; (* A b b r u c h *)
ELSE
	HLI3_CheckChannelValid := TRUE;
	RETURN;
END_IF

END_FUNCTION

// CNC/8 Mis/HLI3_CheckAxisValid
FUNCTION HLI3_CheckAxisValid : BOOL
VAR_INPUT
	nHliAxisIdx: INT;
END_VAR

(* ========================================================= *)
(*    FUN: HLI3_CheckAxisValid                               *)
(* --------------------------------------------------------- *)
(*   Desc: Check if axis ID is valid for HLI access       	 *)
(*   Author: MiB                                             *)
(*   Date: 19.11.2012                                        *)
(*   Rev.: 1.0                                               *)
(* --------------------------------------------------------- *)
(*   Desc: Corrected IF statement (line 17)		 	      	 *)
(*   Author: RCH                                             *)
(*   Date: 16.09.2013                                        *)
(*   Rev.: 1.1                                               *)
(* --------------------------------------------------------- *)
(*   Desc: BugFix: wrong array acces        	 	      	 *)
(*   Author: MiB                                             *)
(*   Date: 05.01.2017                                        *)
(*   Rev.: 1.3                                               *)
(* ========================================================= *)


(* old version *)
(*  
IF (nHliAxisIdx < 0) OR 
	(nHliAxisIdx >= UDINT_TO_INT(gNrAx) ) OR		(* check for axis no *)
    (gpAx[nHliAxisIdx] = 0) 				  (* check for zero pointer *)
THEN
	HLI3_CheckAxisValid:= FALSE;
	RETURN; (* A b b r u c h *)
ELSE
	HLI3_CheckAxisValid := TRUE;
	RETURN;
END_IF *)

(* rev 1.3 *)
IF (nHliAxisIdx < 0) THEN
	HLI3_CheckAxisValid	:= FALSE;
ELSIF (nHliAxisIdx >= UDINT_TO_INT(gNrAx)) THEN
	HLI3_CheckAxisValid	:= FALSE;
ELSIF (gpAx[nHliAxisIdx] = 0 ) THEN
	HLI3_CheckAxisValid	:= FALSE;
ELSE
	HLI3_CheckAxisValid	:= TRUE;
END_IF

END_FUNCTION

// CNC/7 ToolManagement/HLI3_ToolManagement
PROGRAM HLI3_ToolManagement
VAR	
	pToolId: POINTER TO CNC_TOOL_ID;
	pToolReq: POINTER TO CNC_TOOL_REQUEST_IN;
	pToolLife: POINTER TO CNC_TOOL_DATA_IN;
	Rind: ADSRDWRTIND;
	RRes: ADSRDWRTRES;
	bRes: BOOL;
	i: INT;
	nr: DINT;	
	fbRTrigD: R_TRIG;
	fbRTrigOldData: R_TRIG;	
	cnc_channel_nr: UDINT;
	nStateD : INT  := 0;
	nStateT : INT := 0;
	nStateLife: INT := 0;
	
END_VAR

(* ---------------------*----------------------------------|------------------------------------------------------- *)
(* PURPOSE: External Tool Change                                                                                    *)
(*          used for tool change and tool live                                                                      *)
(*                                                                                                                  *)
(* SCOPE:                                                                                                           *)
(*                                                                                                                  *)
(*                                                                                                                  *)
(* REMARKS:                                                                                                         *)
(*                                                                                                                  *)
(*                                                                                                                  *)
(* AUTHOR:              VERSION     DATE                   CHECKED FROM      DATE     STATUS                        *)
(*    MK                1.0         07.05.2003                                                                      *)
(*    MiB               1.1         04.04.2006                                                                      *)
(*    MK                1.2         04.08.2006                                                                      *)
(*	  MiB					1.3			04.12.2006																						    	  *)
(*	  MiB					1.4			19.11.2012          TC3																					  *)
(*	  MiB					1.5			05.03.2015          TC3	  Zusatzparameter P[i]  werden aus der CNC zur PLC in OldTool übertragen		  *)
(*    MiB				2.0			07.09.2017		        TC3   Redesign                                                                                                              *)
(* ---------------------*----------------------------------|------------------------------------------------------- *)

(*
 ATTENTION: These Indications are only sent by the CNC if the CNC channel is configured accordingly:
In the SDA-MDS parammeter list the following parameters must be set:

ext_wzv_vorhanden    1   -> (external tool managment present) Tool requests D<i> are sent TO external tool data manager
einrechnen_mit_t     0/1 -> programming T<i> implies a programmed D<i>
tool_life_to_wzv     1   -> send tool data life parameters TO external tool data manager IF tool is changed.
t_info_to_wzv        1   -> send tool to external tool data manager IF tool is programmed.
d_clear_to_wzv 		 1  ( P-CHAN-00103 hold P Parameter at reset 
flush.d_cmd 		  FAW_D -> implizit #FLUSH WAIR before D Word
*)





(* Init Tool Configuration *)
bRes := FALSE;
Rind();


FOR i := 0 TO HLI_SYS_CH_MAXIDX DO
	IF CNCSystem.Channel[i].ToolData.bResetToolRequest THEN
		IF (UDINT_TO_INT(cnc_channel_nr-1) = i) THEN  // if the last channel is the active channel -> Reset states and send a response
			nStateD := 0;
			nStateT := 0;
			nStateLife := 0;
			RRes.LEN		:= 0;
			RRes.DATAADDR	:= 0;
			RRes.RESULT		:= ADS_RDWRT_IND_UNKNOWN_INDEXGROUP;
			IF (Rind.VALID) THEN 				
				bRes := TRUE;
			END_IF
		END_IF
		CNCSystem.Channel[i].ToolData.bResetToolRequest := FALSE;
	END_IF
END_FOR


IF Rind.VALID THEN
	(* initialize response *)
	RRes.NETID := '';
	RRes.PORT	:= Rind.PORT;
	RRes.INVOKEID := Rind.INVOKEID;

	(* sender channel nr is coded in the invoke id *) (* Kanalnummer zur Zeit nicht benutzt *)
	cnc_channel_nr := RInd.INVOKEID; 
	cnc_channel_nr := cnc_channel_nr AND 16#00FFFFFF; 
	
		
	(* Since there is only one ADSRDWRTIND possible per PLC task *)
	(* all indications have to be handled in one place *)
	(* To distinguish between several possible request types *)
	(* the indexgroup of the ADSRDWRTIND is used *)

	(*----- CNC tool data request with T<i>-----*)
	(* CNC teil den Werkzeugwechsel T<i> (während Programmdekodierung) mit *)
	IF Rind.IDXGRP = ADS_IGRP_TOOL_INFO_WRITE THEN (* 16#80040000  *)

		(* Tool (T) request from CNC *)
		IF (nStateT = 0) THEN
			nStateT := 10;  (* start step chain *)
		END_IF
		IF (HLI3_ToolManagement.T_Command()) THEN
			nStateT := 0;					
			bRes := TRUE;
		END_IF	

	(*----- CNC tool data request with D<i>-----*)
	(* CNC fordert Werkzeuggeometriedaten aufgrund D<i> an *)
	ELSIF Rind.IDXGRP = ADS_IGRP_TOOL_DESC_READ THEN		
		(* Tool data (D) request from CNC *)
		IF (nStateD = 0) THEN
			nStateD := 10;  (* start step chain *)
		END_IF
		IF (HLI3_ToolManagement.D_Command()) THEN
			nStateD := 0;					
			bRes := TRUE;
		END_IF
	

	(*----- CNC tool life -----*)
	(* CNC aktualisiert die Werkzeugstanddaten nach Anwahl eines anderen Werkzeugs T<i> *)
	ELSIF Rind.IDXGRP = ADS_IGRP_TOOL_LIFE_DATA_WRITE THEN
			
		(* ToolLife data from CNC *)
		IF (nStateLife = 0) THEN
			nStateLife := 10;  (* start step chain *)
		END_IF
		IF (HLI3_ToolManagement.ToolLife_Command()) THEN 
			nStateLife := 0;					
			bRes := TRUE;
		END_IF
		
	(* Unknown indexgroup, just send an response *)
	ELSE		
		RRes.LEN		:= 0;
		RRes.DATAADDR	:= 0;
		RRes.RESULT		:= ADS_RDWRT_IND_UNKNOWN_INDEXGROUP;
	END_IF
END_IF


RRes(RESPOND:=bRes);

IF bRes THEN
	RRes(RESPOND:=FALSE);
	Rind(CLEAR:=TRUE);
	Rind(CLEAR:=FALSE);
END_IF

METHOD PUBLIC D_Command : BOOL
VAR_INPUT
END_VAR

CASE nStateD OF 
	0: (* IDLE *)
		D_Command := FALSE;
		
	10:
		pToolReq		:= Rind.DATAADDR;
		IF (CNCSystem.Channel[cnc_channel_nr-1].ToolData.bToolRequest <> TRUE) THEN    
			nStateD := nStateD + 10;
		END_IF
	
	20: (* get actual data for active tool*)
		CNCSystem.Channel[cnc_channel_nr-1].ToolData.nToolRequestID := pToolReq^.act_d_nr.basic;
		CNCSystem.Channel[cnc_channel_nr-1].ToolData.nToolRequestIDSister := pToolReq^.act_d_nr.sister;
		CNCSystem.Channel[cnc_channel_nr-1].ToolData.nToolRequestIDVariant := pToolReq^.act_d_nr.variant;
		CNCSystem.Channel[cnc_channel_nr-1].ToolData.bToolRequest := TRUE;	
		nStateD := nStateD + 10;
		
	30: (* Wait for actual data for active tool *)
	
		IF NOT CNCSystem.Channel[cnc_channel_nr-1].ToolData.bToolRequest THEN	
			CNCSystem.Channel[cnc_channel_nr-1].ToolData.stOldTool := CNCSystem.Channel[cnc_channel_nr-1].ToolData.stActTool;
			CNCSystem.Channel[cnc_channel_nr-1].ToolData.stOldTool.tool_desc.param := pToolReq^.param;	(* get paranmeter array from the cnc*)		
			nStateD := nStateD + 10;
		END_IF
		
	40:  (* send old tool data back to HMI *)
		IF NOT CNCSystem.Channel[cnc_channel_nr-1].ToolData.bOldToolDataExist THEN
			CNCSystem.Channel[cnc_channel_nr-1].ToolData.bOldToolDataExist := TRUE;
			nStateD := nStateD + 10;
		END_IF
		
		
	50: (* Wait until old tool data was read , then get requested data*)
		IF NOT CNCSystem.Channel[cnc_channel_nr-1].ToolData.bOldToolDataExist AND NOT CNCSystem.Channel[cnc_channel_nr-1].ToolData.bToolRequest THEN									
			CNCSystem.Channel[cnc_channel_nr-1].ToolData.nToolRequestID := pToolReq^.id.basic;
			CNCSystem.Channel[cnc_channel_nr-1].ToolData.nToolRequestIDSister := pToolReq^.id.sister;             
			CNCSystem.Channel[cnc_channel_nr-1].ToolData.nToolRequestIDVariant := pToolReq^.id.variant;			
			CNCSystem.Channel[cnc_channel_nr-1].ToolData.bToolRequest := TRUE;	
			nStateD := nStateD + 10;
		END_IF
	
		
	60: (* wait for tool data from HMI *)
		IF NOT CNCSystem.Channel[cnc_channel_nr-1].ToolData.bToolRequest THEN			(* bToolData becomes false, when HMI has send tool data to struture actTool *)
	
				(* Delta verrechnen, da in der CNC nur eine Länge ohne Delta existiert *)
				CNCSystem.Channel[cnc_channel_nr-1].ToolData.stActTool.tool_desc.laenge := CNCSystem.Channel[cnc_channel_nr-1].ToolData.stActTool.laenge + CNCSystem.Channel[cnc_channel_nr-1].ToolData.stActTool.laenge_delta;
				CNCSystem.Channel[cnc_channel_nr-1].ToolData.stActTool.tool_desc.radius := CNCSystem.Channel[cnc_channel_nr-1].ToolData.stActTool.radius + CNCSystem.Channel[cnc_channel_nr-1].ToolData.stActTool.radius_delta;
													
				IF CNCSystem.Channel[cnc_channel_nr-1].ToolData.stActTool.tool_desc.valid THEN				
					CNCSystem.Channel[cnc_channel_nr-1].ToolData.nToolInCnc := CNCSystem.Channel[cnc_channel_nr-1].ToolData.stActTool.tool_desc.tool_id.basic;
					CNCSystem.Channel[cnc_channel_nr-1].ToolData.nToolInCncSister := CNCSystem.Channel[cnc_channel_nr-1].ToolData.stActTool.tool_desc.tool_id.sister;
					CNCSystem.Channel[cnc_channel_nr-1].ToolData.nToolInCncVariant := CNCSystem.Channel[cnc_channel_nr-1].ToolData.stActTool.tool_desc.tool_id.variant;
				END_IF
				
				IF  CNCSystem.Channel[cnc_channel_nr-1].ToolData.DCommand <> 0 THEN		(* if there is a class connected that implements the interface -> call the commmit method and wait until it returns true*)		
					nStateD := nStateD + 10;			
				ELSE
					nStateD := nStateD + 20;
				END_IF			
		END_IF		
		
	70:
		IF CNCSystem.Channel[cnc_channel_nr-1].ToolData.DCommand.Commit(CNCSystem.Channel[cnc_channel_nr-1].ToolData.stActTool) THEN
			CNCSystem.Channel[cnc_channel_nr-1].ToolData.stActTool := CNCSystem.Channel[cnc_channel_nr-1].ToolData.DCommand.Tool;
			nStateD := nStateD + 10;		
		END_IF
		
		
		
	80:
		RRes.LEN		:= SIZEOF(CNCSystem.Channel[cnc_channel_nr-1].ToolData.stActTool.tool_desc);
		RRes.DATAADDR	:= ADR(CNCSystem.Channel[cnc_channel_nr-1].ToolData.stActTool.tool_desc);
		RRes.RESULT		:= ADS_RDWRT_IND_NO_ERROR;			
		nStateD := nStateD + 10;
		
	90: (* ready *)
		D_Command := TRUE;
		
END_CASE
END_METHOD

METHOD PUBLIC T_Command : BOOL
VAR_INPUT
END_VAR



CASE nStateT OF 
	0: (* IDLE *)
		T_Command := FALSE;		
	10:					
		pToolId		:= Rind.DATAADDR;			
		IF (CNCSystem.Channel[cnc_channel_nr-1].ToolData.bToolRequest <> TRUE) THEN    
			nStateT := nStateT + 10;
		END_IF
			
	20:										
		CNCSystem.Channel[cnc_channel_nr-1].ToolData.nToolRequestID := pToolId^.basic;
		CNCSystem.Channel[cnc_channel_nr-1].ToolData.nToolRequestIDSister := pToolId^.sister;
		CNCSystem.Channel[cnc_channel_nr-1].ToolData.nToolRequestIDVariant := pToolId^.variant;		
		CNCSystem.Channel[cnc_channel_nr-1].ToolData.bToolRequest := TRUE;	
		nStateT := nStateT + 10;
		
	30: (* wait for tool data from HMI *)
		IF NOT CNCSystem.Channel[cnc_channel_nr-1].ToolData.bToolRequest THEN		(* bToolData becomes false, when HMI has send tool data to struture actTool *)
				
				CNCSystem.Channel[cnc_channel_nr-1].ToolData.stActT := CNCSystem.Channel[cnc_channel_nr-1].ToolData.stActTool;				
		
				(* Delta verrechnen, da in der CNC nur eine Länge ohne Delta existiert *)
				CNCSystem.Channel[cnc_channel_nr-1].ToolData.stActT.tool_desc.laenge := CNCSystem.Channel[cnc_channel_nr-1].ToolData.stActT.laenge + CNCSystem.Channel[cnc_channel_nr-1].ToolData.stActT.laenge_delta;
				CNCSystem.Channel[cnc_channel_nr-1].ToolData.stActT.tool_desc.radius := CNCSystem.Channel[cnc_channel_nr-1].ToolData.stActT.radius + CNCSystem.Channel[cnc_channel_nr-1].ToolData.stActT.radius_delta;
				CNCSystem.Channel[cnc_channel_nr-1].ToolData.stActT.tool_desc.tool_id.sister_valid := TRUE;
				CNCSystem.Channel[cnc_channel_nr-1].ToolData.stActT.tool_desc.tool_id.variant_valid := TRUE;					
				
				IF  CNCSystem.Channel[cnc_channel_nr-1].ToolData.TCommand <> 0 THEN		(* if there is a class connected that implements the interface -> call the commmit method and wait until it returns true*)		
					nStateT := nStateT + 10;			
				ELSE
					nStateT := nStateT + 20;
				END_IF
		
		END_IF		
		
    40: 
	    IF CNCSystem.Channel[cnc_channel_nr-1].ToolData.TCommand.Commit(CNCSystem.Channel[cnc_channel_nr-1].ToolData.stActT) THEN
			CNCSystem.Channel[cnc_channel_nr-1].ToolData.stActT := CNCSystem.Channel[cnc_channel_nr-1].ToolData.TCommand.Tool;
			nStateT := nStateT + 10;		
		END_IF
		
		
	50:
		RRes.LEN	:= SIZEOF(CNCSystem.Channel[cnc_channel_nr-1].ToolData.stActT.tool_desc.tool_id);
		RRes.DATAADDR	:= ADR(CNCSystem.Channel[cnc_channel_nr-1].ToolData.stActT.tool_desc.tool_id);		
		RRes.RESULT		:= ADS_RDWRT_IND_NO_ERROR;	
		nStateT := nStateT + 10;
		
	60: (* ready *)
		T_Command := TRUE;
		
END_CASE
END_METHOD

METHOD PUBLIC ToolLife_Command : BOOL
VAR_INPUT
END_VAR

CASE nStateLife OF 
	0: (* IDLE *)
		ToolLife_Command := FALSE;		
	10:					

	
		(* CNC writes tool life data *)
		pToolLife := Rind.DATAADDR;
		
		(* no data transmitted in the response *)
		RRes.LEN			:= 0;
		RRes.DATAADDR		:= 0;
		
		IF (CNCSystem.Channel[cnc_channel_nr-1].ToolData.bToolRequest <> TRUE) THEN    
			nStateLife := nStateLife + 10;
		END_IF
				

	20: (* get actual data for  tool*)
		CNCSystem.Channel[cnc_channel_nr-1].ToolData.nToolRequestID := pToolLife^.tool_id.basic;
		CNCSystem.Channel[cnc_channel_nr-1].ToolData.nToolRequestIDSister := pToolLife^.tool_id.sister;
		CNCSystem.Channel[cnc_channel_nr-1].ToolData.nToolRequestIDVariant := pToolLife^.tool_id.variant;
		CNCSystem.Channel[cnc_channel_nr-1].ToolData.bToolRequest := TRUE;	
		nStateLife := nStateLife + 10;
		
	30: (* wait for data, copy to oldTool and update toollife *)
		IF NOT CNCSystem.Channel[cnc_channel_nr-1].ToolData.bToolRequest AND NOT CNCSystem.Channel[cnc_channel_nr-1].ToolData.bOldToolDataExist THEN	
			CNCSystem.Channel[cnc_channel_nr-1].ToolData.stOldTool := CNCSystem.Channel[cnc_channel_nr-1].ToolData.stActTool;
			
			CNCSystem.Channel[cnc_channel_nr-1].ToolData.stOldTool.tool_life.dist_used := CNCSystem.Channel[cnc_channel_nr-1].ToolData.stOldTool.tool_life.dist_used + pToolLife^.dist_used;
			CNCSystem.Channel[cnc_channel_nr-1].ToolData.stOldTool.tool_life.time_used := CNCSystem.Channel[cnc_channel_nr-1].ToolData.stOldTool.tool_life.time_used + pToolLife^.time_used;
			(* Ist das Werkzeug noch gültig ? *)
			IF CNCSystem.Channel[cnc_channel_nr-1].ToolData.stOldTool.dist_max > 0 AND (CNCSystem.Channel[cnc_channel_nr-1].ToolData.stOldTool.tool_life.dist_used > CNCSystem.Channel[cnc_channel_nr-1].ToolData.stOldTool.dist_max) THEN
				CNCSystem.Channel[cnc_channel_nr-1].ToolData.stOldTool.tool_desc.valid := FALSE;
			END_IF
			IF CNCSystem.Channel[cnc_channel_nr-1].ToolData.stOldTool.time_max > 0 AND (CNCSystem.Channel[cnc_channel_nr-1].ToolData.stOldTool.tool_life.time_used > CNCSystem.Channel[cnc_channel_nr-1].ToolData.stOldTool.time_max) THEN
				CNCSystem.Channel[cnc_channel_nr-1].ToolData.stOldTool.tool_desc.valid := FALSE;
			END_IF
			
			IF  CNCSystem.Channel[cnc_channel_nr-1].ToolData.ToolLifeCommand <> 0 THEN		(* if there is a class connected that implements the interface -> call the commmit method and wait until it returns true*)		
				nStateLife := nStateLife + 10;			
			ELSE
				nStateLife := nStateLife + 20;
			END_IF
		END_IF

	40:
		IF CNCSystem.Channel[cnc_channel_nr-1].ToolData.ToolLifeCommand.Commit(CNCSystem.Channel[cnc_channel_nr-1].ToolData.stOldTool) THEN
			CNCSystem.Channel[cnc_channel_nr-1].ToolData.stOldTool := CNCSystem.Channel[cnc_channel_nr-1].ToolData.ToolLifeCommand.Tool;
			nStateLife := nStateLife + 10;		
		END_IF
			
		
	50: 		
		CNCSystem.Channel[cnc_channel_nr-1].ToolData.bOldToolDataExist := TRUE;
		nStateLife := nStateLife + 10;
		
	60:
		IF NOT CNCSystem.Channel[cnc_channel_nr-1].ToolData.bOldToolDataExist THEN
			RRes.RESULT := ADS_RDWRT_IND_NO_ERROR;
			nStateLife := nStateLife + 10;
			// RRes.RESULT := WZV_TOOL_ID_BASIC_INVALID;
		END_IF
		
	
	70: (* ready *)
		ToolLife_Command := TRUE;		
		
	
END_CASE
END_METHOD

END_PROGRAM

// CNC/10 MessagesHandler/CNCErrorDimensionToString
FUNCTION CNCErrorDimensionToString : STRING
VAR_INPUT
	Dimension: DINT;
END_VAR

(* ========================================================= *)
(*    FC: CNCErrorDimensionToString                            *)
(* --------------------------------------------------------- *)
(*   Desc: CNC Error Dimension to String		 			 *)
(*   Author: ISG / TV                                        *)
(*   Date: 23.12.2016                                        *)
(*   Rev.: 1.0                                               *)
(*															 *)
(* ========================================================= *)

CASE Dimension OF
  HLI_NO_DIMENSION:
    CNCErrorDimensionToString := '-';

  HLI_DIM_DIMENSIONSLOS:
    CNCErrorDimensionToString := '';

  HLI_DIM_POSITION:
    CNCErrorDimensionToString := ' [mm or °]';

  HLI_DIM_GESCHWINDIGKEIT:
    CNCErrorDimensionToString := ' [0.001 mm/s or °/s]';

  HLI_DIM_BESCHLEUNIGUNG:
    CNCErrorDimensionToString := ' [mm/s^2 or °/s^2]';

  HLI_DIM_RUCK:
    CNCErrorDimensionToString := ' [mm/s^3 or °/s^3]';

  HLI_DIM_ZEIT:
    CNCErrorDimensionToString := ' [10^-6 s]';

  HLI_DIM_PROZENT:
    CNCErrorDimensionToString :=  ' [0.1 %]';

  HLI_DIM_ADRESSE:
    CNCErrorDimensionToString :=  ' [-]';

  HLI_DIM_INKREMENTE:
    CNCErrorDimensionToString :=  ' [-]';

  HLI_DIM_UMDR_VORSCHUB:
    CNCErrorDimensionToString :=  ' [0.0001 mm/U]';

  HLI_DIM_V_SCHNITT:
    CNCErrorDimensionToString :=  ' [0.001 mm/s]';

  HLI_DIM_WEG_AUFLOESUNG:
    CNCErrorDimensionToString :=  ' [Incr/0.1um]';

  HLI_DIM_INKR_UMDREHUNG:
    CNCErrorDimensionToString :=  ' [Incr/rev]';
    
  HLI_DIM_BYTE:
    CNCErrorDimensionToString :=  ' [-]';

  HLI_DIM_PROPORTIONAL_GAIN:
    CNCErrorDimensionToString :=  ' [0.01/s]';

  HLI_DIM_FREQUENCY:
    CNCErrorDimensionToString :=  ' [Hz]';

  HLI_DIM_LOAD:
    CNCErrorDimensionToString :=  ' [kg or kg*m^2]';
    
  HLI_POSITION_HIGH_RES:
    CNCErrorDimensionToString :=  ' [10^-8 mm or 10^-8 °]';

  HLI_DIM_INCREMENT_HIGH_RES:
    CNCErrorDimensionToString :=  ' [10^-4 Incr]';
	
ELSE
  CNCErrorDimensionToString :=  'unknown dimension ';
  CNCErrorDimensionToString := CONCAT(CNCErrorDimensionToString , DINT_TO_STRING(Dimension));
END_CASE

END_FUNCTION

// CNC/10 MessagesHandler/CNCErrorGetLogAxisId
FUNCTION CNCErrorGetLogAxisId : DINT
VAR_INPUT
	InWert: HLI_WERT_B;
END_VAR
VAR
	PtrUint: POINTER TO UINT := 0;
END_VAR

VAR_IN_OUT
	nLogAxisID : DINT;
END_VAR

(* ========================================================= *)
(*    FC: CNCErrorGetLogAxisId                               *)
(* --------------------------------------------------------- *)
(*   Desc: CNC Error Get LogAxisId from Error Parameters     *)
(*   Author: ISG / TV                                        *)
(*   Date: 04.09.2017                                        *)
(*   Rev.: 1.1                                               *)
(*															 *)
(* ========================================================= *)


IF (InWert.bedeutung = HLI_BEDEUT_LOG_ACHS_NR) THEN
	  PtrUint := ADR(InWert.inhalt);
	  IF (PtrUint^ <> 0) THEN
		  nLogAxisID := PtrUint^;
 	  END_IF
 END_IF

END_FUNCTION

// CNC/10 MessagesHandler/CNCErrorMeaningToString
FUNCTION CNCErrorMeaningToString : STRING
VAR_INPUT
	Bedeut: UDINT;
END_VAR

(* ========================================================= *)
(*    FC: CNCErrorMeaningToString                            *)
(* --------------------------------------------------------- *)
(*   Desc: CNC Error Meaning to String		 			     *)
(*   Author: ISG / TV                                        *)
(*   Date: 23.12.2016                                        *)
(*   Rev.: 1.0                                               *)
(*															 *)
(* ========================================================= *)

CASE Bedeut OF

  HLI_BEDEUT_IGNORE:
    CNCErrorMeaningToString := '';

  HLI_BEDEUT_GRENZ_WERT:
    CNCErrorMeaningToString := 'limit ';

  HLI_BEDEUT_AKT_WERT:
    CNCErrorMeaningToString :='actual ';

  HLI_BEDEUT_FEHL_WERT:
    CNCErrorMeaningToString :='wrong ';

  HLI_BEDEUT_ERWARTET_WERT:
    CNCErrorMeaningToString :='expected ';

  HLI_BEDEUT_KORR_WERT:
    CNCErrorMeaningToString :='adjusted  ';

  HLI_BEDEUT_LOG_ACHS_NR:
    CNCErrorMeaningToString := 'axis ';

  HLI_BEDEUT_ANTR_TYP:
    CNCErrorMeaningToString := 'drivetype ';

  HLI_BEDEUT_LOG_BED_ELEM_NR:
    CNCErrorMeaningToString := 'controlelement ';

  HLI_BEDEUT_ZUSTAND:
    CNCErrorMeaningToString := 'state ';

  HLI_BEDEUT_TRANSITION:
    CNCErrorMeaningToString := 'transition ';

  HLI_BEDEUT_SENDER:
    CNCErrorMeaningToString := 'sender ';

  HLI_BEDEUT_KLASSE:
    CNCErrorMeaningToString := 'class ';

  HLI_BEDEUT_INSTANZ:
    CNCErrorMeaningToString := 'instance ';

  HLI_BEDEUT_IDENT_NR:
    CNCErrorMeaningToString := 'Ident ';

  HLI_BEDEUT_STATUS:
    CNCErrorMeaningToString := 'status ';

  HLI_BEDEUT_RING_NR:
    CNCErrorMeaningToString := 'ring ';

  HLI_BEDEUT_SATZ_NR:
    CNCErrorMeaningToString := 'block ';

  HLI_BEDEUT_MAX_LIMIT:
    CNCErrorMeaningToString := 'max limit ';

  HLI_BEDEUT_MIN_LIMIT:
    CNCErrorMeaningToString := 'min limit ';

  HLI_BEDEUT_START_WERT:
    CNCErrorMeaningToString := 'start ';

  HLI_BEDEUT_ZIEL_WERT:
    CNCErrorMeaningToString := 'destination ';

  HLI_BEDEUT_ERROR_CODE :
    CNCErrorMeaningToString := 'error code ';
ELSE
  CNCErrorMeaningToString := 'unknown meaning: ';
  CNCErrorMeaningToString := CONCAT(CNCErrorMeaningToString , UDINT_TO_STRING(Bedeut));
END_CASE

END_FUNCTION

// CNC/10 MessagesHandler/CNCErrorParameterToString
FUNCTION CNCErrorParameterToString : STRING
VAR_INPUT
	InWert: HLI_WERT_B;
	WertNr: INT;
END_VAR
VAR
	TmpString: STRING;
END_VAR

(* ========================================================= *)
(*    FC: CNCError Parameter ToString                        *)
(* --------------------------------------------------------- *)
(*   Desc: CNC Error Dimension to String		 			 *)
(*   Author: ISG / TV                                        *)
(*   Date: 23.12.2016                                        *)
(*   Rev.: 1.0                                               *)
(*															 *)
(* ========================================================= *)

(* Test ob Element verwendet wird *)

IF InWert.bedeutung <>  HLI_BEDEUT_IGNORE THEN

  CNCErrorParameterToString := '';

  TmpString := CNCErrorMeaningToString(Bedeut := InWert.bedeutung);
  CNCErrorParameterToString := CONCAT(CNCErrorParameterToString, TmpString);

  TmpString := CNCErrorUnionToString(InWert.Inhalt.data, InWert.typ, UDINT_TO_DINT(InWert.dimension), InWert.bedeutung);
  CNCErrorParameterToString := CONCAT(CNCErrorParameterToString, TmpString);

  TmpString := CNCErrorDimensionToString(UDINT_TO_DINT(InWert.dimension));
  CNCErrorParameterToString := CONCAT(CNCErrorParameterToString, TmpString);

ELSE
  CNCErrorParameterToString := '';
END_IF

END_FUNCTION

// CNC/10 MessagesHandler/CNCErrorUnionToString
FUNCTION CNCErrorUnionToString : STRING
VAR_INPUT
	InWert: ARRAY[0..HLI_WERT_B_DATA_MAXIDX] OF BYTE;
	UnionTyp: UDINT;
	Dimension: DINT;
	Bedeut: UDINT;
END_VAR
VAR
	PtrBool: POINTER TO BOOL := 0;
	PtrUSint: POINTER TO USINT := 0;
	PtrSint: POINTER TO SINT := 0;
	PtrUint: POINTER TO UINT := 0;
	PtrInt: POINTER TO INT := 0;
	PtrUDint: POINTER TO UDINT := 0;
	PtrDint: POINTER TO DINT := 0;
	PtrLReal: POINTER TO LREAL := 0;
	PtrString: POINTER TO STRING(HLI_ERR_MSG_STR_LEN) := 0;
	PtrA3Real64: POINTER TO ARRAY[0..2] OF LREAL;
	PtrHighResSgnPos: POINTER TO LINT;
	PtrBitArray32: POINTER TO DWORD;
	PtrBitArray16: POINTER TO WORD;
	TmpUnion: ARRAY[0..HLI_WERT_B_DATA_MAXIDX] OF BYTE;		
	nHliChannelIdx : INT;
	i : INT;
END_VAR

(* ========================================================= *)
(*    FC: CNCError Union ToString                            *)
(* --------------------------------------------------------- *)
(*   Desc: CNC Error Union to String		 			 	 *)
(*   Author: ISG / TV                                        *)
(*   Date: 02.01.2017                                        *)
(*   Rev.: 1.1                                               *)
(*															 *)
(* ========================================================= *)

TmpUnion := InWert;

CASE UnionTyp  OF
  HLI_TYP_NONE:
    CNCErrorUnionToString := '';

  HLI_TYP_BOOLEAN:
    PtrBool := ADR(TmpUnion[0]);
    CNCErrorUnionToString := BOOL_TO_STRING(PtrBool^);

  HLI_TYP_UNS08:
    PtrUSint := ADR(TmpUnion[0]);
    CNCErrorUnionToString := USINT_TO_STRING(PtrUSint^);

  HLI_TYP_SGN08:
    PtrSint := ADR(TmpUnion[0]);
    CNCErrorUnionToString := SINT_TO_STRING(PtrSint^);

  HLI_TYP_UNS16:
    PtrUint := ADR(TmpUnion[0]);	
	IF (bedeut = HLI_BEDEUT_LOG_ACHS_NR) THEN
		CNCErrorUnionToString := UINT_TO_STRING(PtrUint^);
		CNCErrorUnionToString := CONCAT(CNCErrorUnionToString, ', Log. Axis Name : ');
		CNCErrorUnionToString := CONCAT(CNCErrorUnionToString, CNCSystem.LogAxisNo[PtrUint^].strLogName);
						
		IF HLI3_CheckAxisValid(CNCSystem.LogAxisNo[PtrUint^].nHliAxisIdx) THEN
			CNCErrorUnionToString := CONCAT(CNCErrorUnionToString, ', Ch : ');
			CNCErrorUnionToString := CONCAT(CNCErrorUnionToString, UINT_TO_STRING(gpAx[CNCSystem.LogAxisNo[PtrUint^].nHliAxisIdx]^.lr_state.cnc_channel_r));
			
			 nHliChannelIdx  := HLI3_GetHliChannelIdx(gpAx[CNCSystem.LogAxisNo[PtrUint^].nHliAxisIdx]^.lr_state.cnc_channel_r); 
			
			 IF nHliChannelIdx <> -1 THEN 
				 FOR i := 0 TO (HLI_CH_AX_MAX - 1) DO	
					IF PtrUint^ = gpCh[nHliChannelIdx]^.bahn_state.coord_r[i].log_achs_nr_r THEN
						CNCErrorUnionToString := CONCAT(CNCErrorUnionToString, ', Axis Name  : ');																										
						CNCErrorUnionToString := CONCAT(CNCErrorUnionToString, gpCh[nHliChannelIdx]^.bahn_state.coord_r[i].axis_name_r.zeichen);
						EXIT;
					END_IF			
				END_FOR
			 END_IF		
		END_IF 			
	ELSE
    	CNCErrorUnionToString := UINT_TO_STRING(PtrUint^);
	END_IF 
  HLI_TYP_SGN16:
    PtrInt := ADR(TmpUnion[0]);
    CNCErrorUnionToString := INT_TO_STRING(PtrInt^);

  HLI_TYP_UNS32:
    PtrUDint := ADR(TmpUnion[0]);
    CNCErrorUnionToString := UDINT_TO_STRING(PtrUDint^);

  HLI_TYP_SGN32:
    PtrDint := ADR(TmpUnion[0]);
    CNCErrorUnionToString :=  DINT_TO_STRING(PtrDint^);

  HLI_TYP_REAL64:
    PtrLReal := ADR(TmpUnion[0]);
	IF (Dimension = HLI_DIM_POSITION) THEN
    	CNCErrorUnionToString := LREAL_TO_STRING(PtrLReal^/10000.0);
	ELSE			
		CNCErrorUnionToString := LREAL_TO_STRING(PtrLReal^);
	END_IF

  HLI_TYP_STRING:
    PtrString := ADR(TmpUnion[0]);
    CNCErrorUnionToString := PtrString^;

  HLI_TYP_ADRESSE:
    PtrDint := ADR(TmpUnion[0]);
    CNCErrorUnionToString := DINT_TO_STRING(PtrDint^);
    
  HLI_TYP_IGNORE:
    CNCErrorUnionToString := 'ignore';
    
  HLI_TYP_SYMBOL:
    PtrString := ADR(TmpUnion[0]);
    CNCErrorUnionToString := PtrString^;

  HLI_TYP_A3_REAL64:
    PtrA3Real64 := ADR(TmpUnion[0]);
    CNCErrorUnionToString := LREAL_TO_STRING(PtrA3Real64^[0]);
    CNCErrorUnionToString := CONCAT(CNCErrorUnionToString, ', ');
    CNCErrorUnionToString := CONCAT(CNCErrorUnionToString, LREAL_TO_STRING(PtrA3Real64^[1]));
    CNCErrorUnionToString := CONCAT(CNCErrorUnionToString, ', ');
    CNCErrorUnionToString := CONCAT(CNCErrorUnionToString, LREAL_TO_STRING(PtrA3Real64^[2]));

  HLI_TYP_HIGH_RES_SGN_POS:
    PtrHighResSgnPos := ADR(TmpUnion[0]);
    CNCErrorUnionToString := LINT_TO_STRING(PtrHighResSgnPos^);

  HLI_TYP_BITARRAY_32:
    PtrBitArray32 := ADR(TmpUnion[0]);
    CNCErrorUnionToString := DWORD_TO_BINSTR(PtrBitArray32^, 32);
  
  HLI_TYP_BITARRAY_16:
    PtrBitArray32 := ADR(TmpUnion[0]);
    CNCErrorUnionToString := WORD_TO_BINSTR(PtrBitArray16^, 16);
  
ELSE
  CNCErrorUnionToString := 'unknown type: ';
  CNCErrorUnionToString := CONCAT(CNCErrorUnionToString, UDINT_TO_STRING(UnionTyp));
END_CASE

END_FUNCTION

// CNC/8 Mis/HLI3_GetHliChannelIdx
FUNCTION HLI3_GetHliChannelIdx : INT
VAR_INPUT
	nLogChannelId: UINT;
END_VAR
VAR
	i: INT;
END_VAR

(* ================================================================ *)
(*    FUN: HLI3_GetHliChannelIdx                            		*)
(* ---------------------------------------------------------------- *)
(*   Desc: returns the HLIChannelIdx for a given logical Channel id *)
(*   Author: TV                                             		*)
(*   Date: 02.01.2017                                        		*)
(*   Rev.: 1.1                                               		*)
(* ================================================================ *)
HLI3_GetHliChannelIdx := -1;
FOR i := 0 TO UDINT_TO_INT(gNrCh-1) DO	
	IF nLogChannelId = gpCh[i]^.head.channel_nr THEN
		HLI3_GetHliChannelIdx := i;
		RETURN;
	END_IF
	
END_FOR

END_FUNCTION

// CNC/10 MessagesHandler/FB_ChannelError
FUNCTION_BLOCK FB_ChannelError
VAR_INPUT
	nChanIdx: INT;
END_VAR
VAR_OUTPUT
	Valid: BOOL := FALSE;
	/// Identification of channel error 
	ChErrorID: UDINT;
	/// Module name 
	ModuleName: STRING;
	/// Line in source file 
	Line: DINT;
	/// Multiple ID 
	MultipleID: DINT;
	/// Commandable function type 
	CmdFunctionType: DINT;
	/// Identification of the channel 
	ChannelID: DINT;
	/// Communication ID 
	CommuID: DINT;
	/// Cycle counter of CNC 
	CycleCounter: UDINT;
	/// Version name 
	VersionName: STRING;
	/// Remedy class of error 
	RemedyClass: DINT;
	/// Reaction class of error 
	ReactionClass: DINT;
	/// Body type of error 
	BodyType: UDINT;
	/// User message 
	UserMessage: STRING;
	/// Variables of error record body 
	BodyTypeEnum: UDINT;
	NcBlockNr: DINT := 0;
	ProgName: STRING := '';
	FileName: STRING := '';
	FileOffset: UDINT := 0;
	NcBlockOffset: DINT := 0;
	TokenOffset: DINT := 0;
	LogicalPathNr: DINT := 0;
	AddProgInfo: STRING := '';
	CommuMedium: DINT := 0;
	CommuType: UDINT := 0;
	CommuPartner: UDINT := 0;
	FileLine: UDINT := 0;
	ListType: DINT := 0;
	StructName: STRING := '';
	StrValue_1: STRING;
	StrValue_2: STRING;
	StrValue_3: STRING;
	StrValue_4: STRING;
	StrValue_5: STRING;
	MeaningValue_1: STRING;
	MeaningValue_2: STRING;
	MeaningValue_3: STRING;
	MeaningValue_4: STRING;
END_VAR
VAR
	/// Index of channel specific HLI area 	
	pMcError: POINTER TO MC_ERROR;
	pMcError2: POINTER TO MC_ERROR;
	SatzR: HLI_ERROR_SATZ;
	bInitialized: BOOL := FALSE;
	bClear: BOOL := FALSE;
	bUsed: ARRAY[0..CNC_EVENTS_MAXIDX] OF BOOL;
	bToCleanUp: ARRAY[0..CNC_EVENTS_MAXIDX] OF BOOL;
	LogEvent: ARRAY[0..CNC_EVENTS_MAXIDX] OF ADSLOGEVENT;
	FlankeQuit: ARRAY[0..CNC_EVENTS_MAXIDX] OF R_TRIG;
	pLog: POINTER TO ADSLOGEVENT;
	fmtStr: STRING;
	eventId: UDINT;
	i: UDINT;
	idx: UDINT := 0;
	maxWarnings: UINT;
	maxErrors: UINT;
	maxUserEvents: UINT;
	/// Gesamtzahl = Userevents und Errors 
	maxEvents: UINT;
	/// maximal index of an event 
	maxIdxEvents: UINT;
	countWarnings: UINT := 0;
	countErrors: UINT := 0;
	countUserEvents: UINT := 0;
	start_idx: UINT;
	stop_idx: UINT;
	paraPointerArray: ARRAY[0..31] OF POINTER TO UDINT;
	paraIndex: INT;
	pRumpfNcProg: POINTER TO HLI_RUMPF_NC_PROG;
	pRumpfNcProgLr: POINTER TO HLI_RUMPF_NC_PROG_LR;
	pRumpfMds: POINTER TO HLI_RUMPF_MDS;
	pRumpfKommu: POINTER TO HLI_RUMPF_KOMMU;
	pRumpfRamDisk: POINTER TO HLI_RUMPF_RAMDISK;
	pRumpfFile: POINTER TO HLI_RUMPF_FILE;
	pRumpfIntprFile: POINTER TO HLI_RUMPF_INTPR_FILE;
	pRumpfListeBinaer: POINTER TO HLI_RUMPF_LISTE_BINAER;
	pRumpfGcm: POINTER TO HLI_RUMPF_GCM;
	bTcComError: BOOL;
	bAxisErr: BOOL;
	nLogAxisId: DINT;
END_VAR
VAR CONSTANT
	XmlEventId_Rumpf: UDINT := 200;
	XmlEventId_RumpfNcProg: UDINT := 201;
	XmlEventId_RumpfNcProgLr: UDINT := 202;
	XmlEventId_RumpfMds: UDINT := 203;
	XmlEventId_RumpfKommu: UDINT := 204;
	XmlEventId_RumpfRamDisk: UDINT := 205;
	XmlEventId_RumpfFile: UDINT := 206;
	XmlEventId_RumpfIntprFile: UDINT := 207;
	XmlEventId_RumpfListeBinaer: UDINT := 208;
	XmlEventId_RumpfGcm: UDINT := 209;
	CNC_SOURCE_ID_BASE: UDINT := 551;
	CNC_USER_SOURCE_ID_BASE: UDINT := 651;
	MAX_CNC_ERRORS: UDINT := 49;
	MAX_CNC_USER_EVENTS: UDINT := 49;
	/// MAX_CNC_ERRORS + MAX_CNC_USER_EVENTS 
	MAX_CNC_EVENTS: UDINT := 98;
	/// MAX_CNC_EVENTS - 1 
	CNC_EVENTS_MAXIDX: UDINT := 97;
	ERR_BAHN_ONLINE_TRC_CALCULATION: UDINT := 50689;
	ERR_ID_REPORT_CNC_RESET: UDINT := 270076;
	ERR_ID_KIN_TRAFO_CONFIG: UDINT := 292030;
	ERR_ID_KIN_TRAFO_INIT: UDINT := 292031;
	ERR_ID_KIN_TRAFO_FORWARD: UDINT := 292032;
	ERR_ID_KIN_TRAFO_BACKWARD: UDINT := 292033;
END_VAR

(* ========================================================= *)
(*    FB: FB_ChannelError                               	 *)
(* --------------------------------------------------------- *)
(*   Desc: FB transfers CNC Errors to the Event Logger		 *)
(*   Author: ISG / TV                                        *)
(*   Date: 04.09.2017                                        *)
(*   Rev.: 1.5                                               *)
(*															 *)
(* ========================================================= *)

(* check for channel no *)
IF NOT HLI3_CheckChannelValid(nChannel := nChanIdx) THEN
	RETURN;
END_IF

(* check for zero pointer *)
IF gpCh[nChanIdx] = 0 THEN
  RETURN;
END_IF

(* check for zero pointer, first channel is necessary for axis errors (Position controller errors) *)
IF gpCh[0] = 0 THEN
  RETURN;
END_IF

pMcError := ADR(gpCh[nChanIdx]^.mc_error);
SatzR    := pMcError^.satz_r;

IF bInitialized = FALSE THEN
  pMcError^.enable_w := TRUE;    (* enable control unit for error messages *) 
  bInitialized  := TRUE;
  maxErrors     := UDINT_TO_UINT(MAX_CNC_ERRORS / gNrCh);
  maxWarnings   := maxErrors / 5;
  maxUserEvents := UDINT_TO_UINT(MAX_CNC_USER_EVENTS / gNrCh);
  maxEvents     := maxUserEvents + maxErrors;

  maxIdxEvents := (maxEvents - 1);
  FOR i := 0 TO maxIdxEvents DO
    (* ----------------------------------------- *)
    (* initialize fixed elements of event        *)
    (* ----------------------------------------- *)
    pLog := ADR( LogEvent[i] );
    pLog^.NETID := '';      (* Local Computer *)
    pLog^.PORT:= 110;       (* Event Logger *)
    pLog^.TMOUT:= t#10s;
    pLog^.EventConfigData.Prio         := TCEVENTPRIO_IMPLICIT;
    pLog^.EventConfigData.ProgId       := 'TcEventFormatter.TcXmlFormatter';
    pLog^.EventConfigData.Flags        := TCEVENTFLAG_SRCID OR TCEVENTFLAG_LOG;
    pLog^.EventConfigData.SourceString := '';
    pLog^.EventConfigData.StreamType   := TCEVENTSTREAM_NORMAL;

    IF i < maxErrors THEN
      (* SourceID: 550 error texts, [ 551,  599] for single CNC error messages *)
      pLog^.EventConfigData.SourceId := CNC_SOURCE_ID_BASE + i + (DINT_TO_UINT(nChanIdx)*maxErrors);
    ELSE
      (* SourceID: 650 user error texts, [ 651,  699] for single CNC user error messages "ERROR[]" *)
      pLog^.EventConfigData.SourceId := CNC_USER_SOURCE_ID_BASE + i-maxErrors + (DINT_TO_UINT(nChanIdx)*maxUserEvents);
    END_IF

    FlankeQuit[i](CLK :=  pLog^.Quit);
  END_FOR
END_IF



(* -------------------------------------------------------------------------*)
(* test if events which have been reported shall be cleared again           *)
(* -------------------------------------------------------------------------*)
IF bClear THEN
  bClear := FALSE;
  countWarnings := 0;
  countErrors := 0;
  countUserEvents := 0;
  FOR i := 0 TO maxIdxEvents DO
    IF bToCleanup[i] = FALSE AND bUsed[i] THEN
      bToCleanup[i] := TRUE;
    END_IF
  END_FOR
END_IF


(* -------------------------------------------------------------------------*)
(* check for new error message                                              *)
(* -------------------------------------------------------------------------*)

(* Output for position controller errors is gpCh[0]^ *)
IF gpCh[0]^.mc_error.semaphor_rw THEN	
	SatzR := gpCh[0]^.mc_error.satz_r;		
	bAxisErr := TRUE;				
END_IF

IF (pMcError^.semaphor_rw  OR bAxisErr)  THEN

 	IF  SatzR.kopf.cnc_channel > 0 THEN 
  		IF (SatzR.kopf.cnc_channel-1 <> INT_TO_UINT(nChanIdx)) THEN	  
			bAxisErr := FALSE;		
    	RETURN;
	END_IF
  END_IF
  
  (* Initialize output variables that depend on error body type *)
  NcBlockNr      := 0;
  ProgName       := '';
  FileName       := '';
  FileOffset     := 0;
  NcBlockOffset  := 0;
  TokenOffset    := 0;
  LogicalPathNr  := 0;
  AddProgInfo    := '';

  CommuMedium    := 0;
  CommuType      := 0;
  CommuPartner   := 0;

  FileLine       := 0;
  ListType       := 0;
  StructName     := '';

  StrValue_1     := '';
  StrValue_2     := '';
  StrValue_3     := '';
  StrValue_4     := '';
  StrValue_5     := '';

  MeaningValue_1 := '';
  MeaningValue_2 := '';
  MeaningValue_3 := '';
  MeaningValue_4 := '';
  
  nLogAxisId   := 0;


  eventId := SatzR.kopf.error_id;

  (*------------------------------------------------------------------*)
  (* automatic clear old events if CNC reports reset                  *)
  (*------------------------------------------------------------------*)
  IF eventId = ERR_ID_REPORT_CNC_RESET THEN
	  	IF bAxisErr THEN 
    		gpCh[0]^.mc_error.semaphor_rw := FALSE;
			bAxisErr := FALSE;
		ELSE
			pMcError^.semaphor_rw := FALSE;		
		END_IF
	
    bClear := TRUE;
    RETURN;
  END_IF

  
  (*------------------------------------------------------------------*)
  (* TcCom: kinematic transformation, map util_error_id to error_id   *)
  (*------------------------------------------------------------------*)
  IF    eventId = ERR_ID_KIN_TRAFO_CONFIG
     OR eventId = ERR_ID_KIN_TRAFO_INIT  
     OR eventId = ERR_ID_KIN_TRAFO_FORWARD
     OR eventId = ERR_ID_KIN_TRAFO_BACKWARD
   OR eventId = ERR_BAHN_ONLINE_TRC_CALCULATION
  THEN
    eventId := SatzR.kopf.util_error_id;
    bTcComError := TRUE;
  ELSE
    bTcComError := FALSE;
  END_IF
   

  (*-------------------------------*)
  (* search unused event           *)
  (*-------------------------------*)
  IF eventId <= 1000 OR bTcComError THEN
    countUserEvents := countUserEvents + 1;
    start_idx       := maxErrors;
    stop_idx        := maxErrors + maxUserEvents - 1;
  ELSE
    (*------------------------------------------------------------------*)
    (* check maximum number of active warnings                          *)
    (*------------------------------------------------------------------*)
    IF SatzR.kopf.behebungs_klasse < 2 THEN
      IF countWarnings > maxWarnings THEN
		  IF (bAxisErr) THEN
			  	gpCh[0]^.mc_error.semaphor_rw := FALSE;
				bAxisErr := FALSE;
		  ELSE	
				pMcError^.semaphor_rw := FALSE;	  
		  END_IF
        
        RETURN;  (* dismiss further warning *)
      END_IF
      countWarnings:= countWarnings + 1;
    END_IF

    countErrors := countErrors + 1;
    start_idx   := 0;
    stop_idx    := maxErrors - 1;
  END_IF

  FOR i := start_idx TO stop_idx DO
    IF bUsed[i] = FALSE THEN
      EXIT;
    END_IF
  END_FOR

  IF i > stop_idx THEN
    (*------------------------------------------------------------------*)
    (* overflow -> dismiss actual message, wait for reset               *)
    (*------------------------------------------------------------------*)
	IF (bAxisErr) THEN
		gpCh[0]^.mc_error.semaphor_rw := FALSE;
		bAxisErr := FALSE;
	ELSE	
		pMcError^.semaphor_rw := FALSE;	  
	END_IF	
    RETURN;
  END_IF
  idx := i;


  bUsed[idx] := TRUE;
  pLog := ADR( LogEvent[idx] );

  (* Initialisierungen fuer jeden Aufruf *)
  paraIndex := 0;

  (*
    TCEVENTCLASS_NONE        := 0,  No class
    TCEVENTCLASS_MAINTENANCE := 1,  Maintenance hint
    TCEVENTCLASS_MESSAGE     := 2,  Message
    TCEVENTCLASS_HINT        := 3,  Hint
    TCEVENTCLASS_STATEINFO   := 4,  State information
    TCEVENTCLASS_INSTRUCTION := 5,  Instruction
    TCEVENTCLASS_WARNING     := 6,  Warning
    TCEVENTCLASS_ALARM       := 7,  Alarm
    TCEVENTCLASS_PARAMERROR
  *)

  IF SatzR.kopf.behebungs_klasse < 2 THEN
    pLog^.EventConfigData.Class := TCEVENTCLASS_WARNING;
    pLog^.EventConfigData.bQuitRequired := FALSE;  (* Hasn't to acknowledge the event *)
  ELSE
    pLog^.EventConfigData.bQuitRequired := TRUE;  (* Has to acknowledge the event *)
    IF SatzR.kopf.behebungs_klasse < 7 THEN
      pLog^.EventConfigData.Class := TCEVENTCLASS_ALARM;
    ELSE
      pLog^.EventConfigData.Class := TCEVENTCLASS_PARAMERROR;
    END_IF
  END_IF
  pLog^.EventConfigData.Id := XmlEventId_Rumpf;

  (*------------------------------------------------------------------*)
  (* parameters 1 - 13 are content independent                        *)
  (*------------------------------------------------------------------*)
  fmtStr := '%d%d%d%d%s%d%d%d%d%d%s%d%s';  (* a string *)

  (* If ChErrorID has a link to a sub string (other EventId and SourceId)  *)
  (* a string is build of following syntax: '[SxEy]' with x as SourceId and y as EventId *)
  (* in TcCncError.xml x alsways has value 2 and y is the ChErrorID of the CNC *)
  (* ----------------------------------------------------*)
  (* User specific error message                         *)
  (* ----------------------------------------------------*)
  IF eventId <= 1000 OR bTcComError THEN
    UserMessage   := '[S650E'; (* sub string from SourceId 550 (see TcCncUserEvents.xml) and EventId 'eventId' *)
  ELSE
    UserMessage   := '[S550E'; (* sub string from SourceId 2 (see TcCncError.xml) and EventId 'eventId' *)
  END_IF
  UserMessage     := CONCAT(UserMessage, UDINT_TO_STRING(eventId));
  UserMessage     := CONCAT(UserMessage, ']');

  ChErrorID       := eventId;
  ChannelID       := SatzR.kopf.cnc_channel;
  RemedyClass     := SatzR.kopf.behebungs_klasse;
  ReactionClass   := SatzR.kopf.reaktions_klasse;
  ModuleName      := SatzR.kopf.modul_name.zeichen;
  Line            := SatzR.kopf.line;
  MultipleID      := SatzR.kopf.multiple_id;
  CmdFunctionType := SatzR.kopf.bf_type;

  CommuID         := SatzR.kopf.kommu_id;
  CycleCounter    := SatzR.kopf.fb_zeitangabe.zykl_counter;
  VersionName     := SatzR.kopf.version_name.zeichen;
  BodyType        := SatzR.kopf.rumpf_typ;

  paraPointerArray[paraIndex] := ADR(ChErrorID);
  paraIndex := paraIndex + 1;
  paraPointerArray[paraIndex] := ADR(ChannelID);
  paraIndex := paraIndex + 1;
  paraPointerArray[paraIndex] := ADR(RemedyClass);
  paraIndex := paraIndex + 1;
  paraPointerArray[paraIndex] := ADR(ReactionClass);
  paraIndex := paraIndex + 1;
  paraPointerArray[paraIndex] := ADR(ModuleName);
  paraIndex := paraIndex + 1;
  paraPointerArray[paraIndex] := ADR(Line);
  paraIndex := paraIndex + 1;
  paraPointerArray[paraIndex] := ADR(MultipleID);
  paraIndex := paraIndex + 1;
  paraPointerArray[paraIndex] := ADR(CmdFunctionType);
  paraIndex := paraIndex + 1;
  paraPointerArray[paraIndex] := ADR(CommuID);
  paraIndex := paraIndex + 1;
  paraPointerArray[paraIndex] := ADR(CycleCounter);
  paraIndex := paraIndex + 1;
  paraPointerArray[paraIndex] := ADR(VersionName);
  paraIndex := paraIndex + 1;
  paraPointerArray[paraIndex] := ADR(BodyType);
  paraIndex := paraIndex + 1;
  paraPointerArray[paraIndex] := ADR(UserMessage);
  paraIndex := paraIndex + 1;


  (*------------------------------------------------------------------------*)
  (* Append values and meaning of values.                                   *)
  (*------------------------------------------------------------------------*)
  
  StrValue_1 := CNCErrorParameterToString(SatzR.rumpf.wert_1, 1);
  StrValue_2 := CNCErrorParameterToString(SatzR.rumpf.wert_2, 2);
  StrValue_3 := CNCErrorParameterToString(SatzR.rumpf.wert_3, 3);
  StrValue_4 := CNCErrorParameterToString(SatzR.rumpf.wert_4, 4);
  StrValue_5 := CNCErrorParameterToString(SatzR.rumpf.wert_5, 5);  
   
  CNCErrorGetLogAxisId(SatzR.rumpf.wert_1,nLogAxisId);
  CNCErrorGetLogAxisId(SatzR.rumpf.wert_2,nLogAxisId);
  CNCErrorGetLogAxisId(SatzR.rumpf.wert_3,nLogAxisId);
  CNCErrorGetLogAxisId(SatzR.rumpf.wert_4,nLogAxisId);
  CNCErrorGetLogAxisId(SatzR.rumpf.wert_5,nLogAxisId);
  
  CNCSystem.LogAxisNo[nLogAxisId].nCNCErrorID :=  ChErrorID;
     
  paraPointerArray[paraIndex] := ADR(StrValue_1);
  paraIndex := paraIndex + 1;
  paraPointerArray[paraIndex] := ADR(StrValue_2);
  paraIndex := paraIndex + 1;
  paraPointerArray[paraIndex] := ADR(StrValue_3);
  paraIndex := paraIndex + 1;
  paraPointerArray[paraIndex] := ADR(StrValue_4);
  paraIndex := paraIndex + 1;
  paraPointerArray[paraIndex] := ADR(StrValue_5);
  paraIndex := paraIndex + 1;

  fmtStr := CONCAT(fmtStr, '%s%s%s%s%s');

  MeaningValue_1 := WertToString(SatzR.rumpf.kennung_1, 1);
  MeaningValue_2 := WertToString(SatzR.rumpf.kennung_2, 2);
  MeaningValue_3 := WertToString(SatzR.rumpf.kennung_3, 3);
  MeaningValue_4 := WertToString(SatzR.rumpf.kennung_4, 4);

  paraPointerArray[paraIndex] := ADR(MeaningValue_1);
  paraIndex := paraIndex + 1;
  paraPointerArray[paraIndex] := ADR(MeaningValue_2);
  paraIndex := paraIndex + 1;
  paraPointerArray[paraIndex] := ADR(MeaningValue_3);
  paraIndex := paraIndex + 1;
  paraPointerArray[paraIndex] := ADR(MeaningValue_4);
  paraIndex := paraIndex + 1;

  fmtStr := CONCAT(fmtStr, '%s%s%s%s');



  BodyTypeEnum := SatzR.kopf.rumpf_typ;

  (*-------------------------------------------------------------------------*)
  (*       HLI_RUMPF_TYP_NC_PROG                                             *)
  (*-------------------------------------------------------------------------*)
  IF BodyTypeEnum = HLI_RUMPF_TYP_NC_PROG THEN
    pLog^.EventConfigData.Id := XmlEventId_RumpfNcProg;

    pRumpfNcProg := ADR(SatzR.rumpf.maske);

    (* Assign error body data to output variables *)
    NcBlockNr     := pRumpfNcProg^.satz_nr;
    ProgName      := pRumpfNcProg^.prog_name.zeichen;
    FileName      := pRumpfNcProg^.file_name.zeichen;
    FileOffset    := pRumpfNcProg^.fileoffset;
    NcBlockOffset := pRumpfNcProg^.satzoffset;
    TokenOffset   := pRumpfNcProg^.tokenoffset;
    LogicalPathNr := pRumpfNcProg^.log_pfad_nr;
    AddProgInfo   := ''; //  pRumpfNcProg^.add_prog_info.zeichen;

    (* Assign address of data to parameter array of the event *)
    paraPointerArray[paraIndex] := ADR(NcBlockNr);
    paraIndex := paraIndex + 1;
    paraPointerArray[paraIndex] := ADR(ProgName);
    paraIndex := paraIndex + 1;
    paraPointerArray[paraIndex] := ADR(FileName);
    paraIndex := paraIndex + 1;
    paraPointerArray[paraIndex] := ADR(FileOffset);
    paraIndex := paraIndex + 1;
    paraPointerArray[paraIndex] := ADR(NcBlockOffset);
    paraIndex := paraIndex + 1;
    paraPointerArray[paraIndex] := ADR(TokenOffset);
    paraIndex := paraIndex + 1;
    paraPointerArray[paraIndex] := ADR(LogicalPathNr);
    paraIndex := paraIndex + 1;
    paraPointerArray[paraIndex] := ADR(AddProgInfo);
    paraIndex := paraIndex + 1;

    (* Add format string for error messages out of NC programs *)
    fmtStr := CONCAT(fmtStr, '%d%s%s%d%d%d%d%s');
  (*-------------------------------------------------------------------------*)
  (*       HLI_RUMPF_TYP_NC_PROG_LR                                          *)
  (*-------------------------------------------------------------------------*)
  ELSIF BodyTypeEnum = HLI_RUMPF_TYP_NC_PROG_LR THEN
    pLog^.EventConfigData.Id := XmlEventId_RumpfNcProgLR;

    pRumpfNcProgLr := ADR(SatzR.rumpf.maske);

    LogicalPathNr  := pRumpfNcProgLr^.log_pfad_nr;
    ProgName       := pRumpfNcProgLr^.prog_name.zeichen;
    FileName       := pRumpfNcProgLr^.file_name.zeichen;
    NcBlockNr      := pRumpfNcProgLr^.satz_nr;
    AddProgInfo    := ''; //pRumpfNcProgLr^.add_prog_info.zeichen;

    paraPointerArray[paraIndex] := ADR(NcBlockNr);
    paraIndex := paraIndex + 1;
    paraPointerArray[paraIndex] := ADR(ProgName);
    paraIndex := paraIndex + 1;
    paraPointerArray[paraIndex] := ADR(FileName);
    paraIndex := paraIndex + 1;
    paraPointerArray[paraIndex] := ADR(LogicalPathNr);
    paraIndex := paraIndex + 1;
    paraPointerArray[paraIndex] := ADR(AddProgInfo);
    paraIndex := paraIndex + 1;

    fmtStr := CONCAT(fmtStr, '%d%s%s%d%s');
  (*-------------------------------------------------------------------------*)
  (*       HLI_RUMPF_TYP_MDS                                                 *)
  (*-------------------------------------------------------------------------*)
  ELSIF BodyTypeEnum = HLI_RUMPF_TYP_MDS THEN
    pLog^.EventConfigData.Id := XmlEventId_RumpfMds;

    pRumpfMds     := ADR(SatzR.rumpf.maske);

    LogicalPathNr := pRumpfMds^.listen_typ;
    ProgName      := pRumpfMds^.strukt_name.zeichen;

    paraPointerArray[paraIndex] := ADR(LogicalPathNr);
    paraIndex := paraIndex + 1;
    paraPointerArray[paraIndex] := ADR(ProgName);
    paraIndex := paraIndex + 1;

    fmtStr := CONCAT(fmtStr, '%d%s');
  (*-------------------------------------------------------------------------*)
  (*       HLI_RUMPF_TYP_KOMMU                                               *)
  (*-------------------------------------------------------------------------*)
  ELSIF BodyTypeEnum = HLI_RUMPF_TYP_KOMMU THEN
    pLog^.EventConfigData.Id := XmlEventId_RumpfKommu;

    pRumpfKommu  := ADR(SatzR.rumpf.maske);

    CommuMedium  := pRumpfKommu^.Medium;
    CommuType    := pRumpfKommu^.Typ;
    CommuPartner := pRumpfKommu^.Partner;

    paraPointerArray[paraIndex] := ADR(CommuMedium);
    paraIndex := paraIndex + 1;
    paraPointerArray[paraIndex] := ADR(CommuType);
    paraIndex := paraIndex + 1;
    paraPointerArray[paraIndex] := ADR(CommuPartner);
    paraIndex := paraIndex + 1;

    fmtStr := CONCAT(fmtStr, '%d%d%d');
  (*-------------------------------------------------------------------------*)
  (*       HLI_RUMPF_TYP_RAMDISK                                             *)
  (*-------------------------------------------------------------------------*)
  ELSIF BodyTypeEnum = HLI_RUMPF_TYP_RAMDISK THEN
    pLog^.EventConfigData.Id := XmlEventId_RumpfRamDisk;

    pRumpfRamDisk := ADR(SatzR.rumpf.maske);

    CommuMedium   := pRumpfRamDisk^.medium;
    CommuType     := pRumpfRamDisk^.typ;
    CommuPartner  := pRumpfRamDisk^.partner;
    FileName      := pRumpfRamDisk^.file_name.zeichen;
    FileOffset    := pRumpfRamDisk^.fileoffset;

    paraPointerArray[paraIndex] := ADR(CommuMedium);
    paraIndex := paraIndex + 1;
    paraPointerArray[paraIndex] := ADR(CommuType);
    paraIndex := paraIndex + 1;
    paraPointerArray[paraIndex] := ADR(CommuPartner);
    paraIndex := paraIndex + 1;
    paraPointerArray[paraIndex] := ADR(FileName);
    paraIndex := paraIndex + 1;
    paraPointerArray[paraIndex] := ADR(FileOffset);
    paraIndex := paraIndex + 1;

    fmtStr := CONCAT(fmtStr, '%d%d%d%s%d');
  (*-------------------------------------------------------------------------*)
  (*       HLI_RUMPF_TYP_FILE                                                *)
  (*-------------------------------------------------------------------------*)
  ELSIF BodyTypeEnum = HLI_RUMPF_TYP_FILE THEN
    pLog^.EventConfigData.Id := XmlEventId_RumpfFile;

    pRumpfFile := ADR(SatzR.rumpf.maske);

    FileName   := pRumpfFile^.file_name.zeichen;
    FileOffset := pRumpfFile^.fileoffset;

    paraPointerArray[paraIndex] := ADR(FileName);
    paraIndex := paraIndex + 1;
    paraPointerArray[paraIndex] := ADR(FileOffset);
    paraIndex := paraIndex + 1;

    fmtStr := CONCAT(fmtStr, '%s%d');
  (*-------------------------------------------------------------------------*)
  (*       HLI_RUMPF_TYP_INTPR_FILE                                          *)
  (*-------------------------------------------------------------------------*)
  ELSIF BodyTypeEnum = HLI_RUMPF_TYP_INTPR_FILE THEN
    pLog^.EventConfigData.Id := XmlEventId_RumpfIntprFile;

    pRumpfIntprFile := ADR(SatzR.rumpf.maske);

    FileName   := pRumpfIntprFile^.file_name.zeichen;
    FileOffset := pRumpfIntprFile^.fileoffset;
    FileLine   := pRumpfIntprFile^.file_line_number;
    ListType   := pRumpfIntprFile^.listen_typ;
    StructName := pRumpfIntprFile^.strukt_name.zeichen;

    paraPointerArray[paraIndex] := ADR(FileName);
    paraIndex := paraIndex + 1;
    paraPointerArray[paraIndex] := ADR(FileOffset);
    paraIndex := paraIndex + 1;
    paraPointerArray[paraIndex] := ADR(FileLine);
    paraIndex := paraIndex + 1;
    paraPointerArray[paraIndex] := ADR(ListType);
    paraIndex := paraIndex + 1;
    paraPointerArray[paraIndex] := ADR(StructName);
    paraIndex := paraIndex + 1;

    fmtStr := CONCAT(fmtStr, '%s%d%d%d%s');
  (*-------------------------------------------------------------------------*)
  (*       HLI_RUMPF_TYP_LISTE_BINAER                                        *)
  (*-------------------------------------------------------------------------*)
  ELSIF BodyTypeEnum = HLI_RUMPF_TYP_LISTE_BINAER THEN
    pLog^.EventConfigData.Id := XmlEventId_RumpfListeBinaer;

    pRumpfListeBinaer := ADR(SatzR.rumpf.maske);

    StructName:=pRumpfListeBinaer^.strukt_name.zeichen;

    paraPointerArray[paraIndex] := ADR(StructName);
    paraIndex := paraIndex + 1;

    fmtStr := CONCAT(fmtStr, '%s');
  (*-------------------------------------------------------------------------*)
  (*       HLI_RUMPF_TYP_GCM                                                 *)
  (*-------------------------------------------------------------------------*)
  ELSIF BodyTypeEnum = HLI_RUMPF_TYP_GCM THEN
    pLog^.EventConfigData.Id := XmlEventId_RumpfGcm;

    pRumpfGcm := ADR(SatzR.Rumpf.Maske);

    ProgName:=pRumpfGcm^.Token.zeichen;
    FileName:=pRumpfGcm^.FileName.zeichen;

    paraPointerArray[paraIndex] := ADR(ProgName);
    paraIndex := paraIndex + 1;
    paraPointerArray[paraIndex] := ADR(FileName);
    paraIndex := paraIndex + 1;

    fmtStr := CONCAT(fmtStr, '%s%s');
  END_IF

  (*------------------------------------------------------------------------*)
  (* Set values at input pins of FB                                         *)
  (*------------------------------------------------------------------------*)
  pLog^.EventDataAddress:= ADR(paraPointerArray);
  pLog^.EventDataLength:= 0;
  pLog^.fbCleanUp  := FALSE;
  pLog^.EventQuit  := FALSE;

  pLog^.EventConfigData.DataFormatStrAddress := ADR(fmtStr);

  (*------------------------------------------------------------------------*)
  (* report error message to event logger                                   *)
  (*------------------------------------------------------------------------*)
  pLog^(Event := TRUE);

  (* Notify at output that a error essage occurred *)
  Valid := TRUE;

  (* Acknowledge error message *)
 	IF (bAxisErr) THEN
		gpCh[0]^.mc_error.semaphor_rw := FALSE;
		bAxisErr := FALSE;
	ELSE	
		pMcError^.semaphor_rw := FALSE;	  
	END_IF
ELSE
  Valid := FALSE;
END_IF

(* by default : no error message is present, first search for error messages *)
FOR i := 0 TO maxIdxEvents DO
  (*-------------------------------------------------------------------------*)
  (*       clear event                                                       *)
  (*-------------------------------------------------------------------------*)
  IF bToCleanup[i] THEN
    pLog := ADR( LogEvent[i] );
    pLog^();

    IF pLog^.EventState=TCEVENTSTATE_SIGNALED THEN
      pLog^( Event:=FALSE);
    ELSIF pLog^.EventState=TCEVENTSTATE_RESET THEN
      pLog^( EventQuit:= TRUE);
    ELSIF pLog^.EventState=TCEVENTSTATE_CONFIRMED OR pLog^.EventState=TCEVENTSTATE_INVALID THEN
      (*pLog^( FbCleanup:= TRUE); bugfix 12.7.2005*)
      bUsed[i]     := FALSE;
      bToCleanup[i] := FALSE;
    END_IF;
  (*-------------------------------------------------------------------------*)
  (*       report event                                                      *)
  (*-------------------------------------------------------------------------*)
  ELSIF bUsed[i] THEN
    pLog := ADR( LogEvent[i] );
    pLog^();

    (* IF pLog^.EventConfigData.bQuitRequired = FALSE THEN
      FlankeQuit[i](CLK :=  pLog^.Quit);
      IF FlankeQuit[i].Q = TRUE THEN
        bUsed[i] := FALSE;
        QuitCount := QuitCount + 1;
      END_IF
    END_IF*)
  END_IF
END_FOR

END_FUNCTION_BLOCK

// CNC/11 Util/F_GRAYCODE_TO_UINT
FUNCTION F_GRAYCODE_TO_UINT : UINT
VAR_INPUT
	byGraycodeSwitches	: BYTE;
END_VAR
VAR
	nLoopCount				: INT;
	byResult					: BYTE;
	bySwitches				: BYTE;
END_VAR

bySwitches			:= byGraycodeSwitches;
byResult				:= 0;

FOR nLoopCount := 0 TO 31 DO
	byResult 		:= byResult XOR bySwitches;
	bySwitches		:= SHR(bySwitches, 1);
END_FOR

F_GRAYCODE_TO_UINT	:= BYTE_TO_UINT(byResult);

END_FUNCTION

// CNC/11 Util/FB_CNCWriteParameter
///*********************************************************************************************************
///NAME.......................:		FB_CNCWriteParameter
///DATUM....................:		08.12.2017
///AUTOR....................:		Thomas Voß
///VERSION................:			1.4
///
///Description.: 	The function block allows to write cnc parameters to the CNC kernel.					
///**********************************************************************************************************
FUNCTION_BLOCK FB_CNCWriteParameter
VAR_INPUT
	/// Channel Id	
	nLogChannelID : UINT;
	/// log. Axis Id  
	nLogAxisId: UINT;
	bExecute: BOOL;
	/// numbers of parameters 
	nNumParameters: INT;
	/// Parameter type
	eParameterType: E_CNCParameterTypes;
	/// Windows temp file for sub lists
	strTempPath: STRING;
	stParameter: ARRAY[0..199] OF ST_CNCParameter;
END_VAR
VAR_OUTPUT
	bBusy: BOOL;
	bError: BOOL;
	nErrorID: INT;
END_VAR

VAR
	fbOnTrigger: R_TRIG;
	Step: UDINT;
	FbAdsWrite: ADSWRITE;
	strParameterLine: STRING(255);
	strFileName: STRING(255);
	strHeader: STRING(255);
	TimeOut: TON;
	m: DINT;
	/// Text To File 
	fbFileOpen: FB_FileOpen;
	fbFileRead: FB_FileRead;
	fbFilePuts: FB_FilePuts;
	fbFileClose: FB_FileClose;
	hFileOutput: UINT := 0;
END_VAR
VAR CONSTANT
	nMaxParameters: INT := 200;
	/// Ads Interface 
	nAdsPortNumber: UINT := 553;
	nAdsIndexGroup: UDINT := 16#20100;
	nAdsIndexGroupAxisParameter: UDINT := 16#20200;
	nAdsIndexOffsetlogAxisNumber: UDINT := 16#37;
	nAdsIndexOffsetChannelParameter: UDINT := 16#34;	
	nAdsIndexOffsetAxisParameter: UDINT := 16#18;
	nAdsIndexOffsetZeroOffsets: UDINT := 16#2E;
	nAdsIndexOffsetToolParameter: UDINT := 16#30;
	nAdsIndexOffsetClampPosition: UDINT := 16#32;
	nAdsIndexOffsetCompensationTable: UDINT := 16#39;
	/// Time Out Error 
	ErrID_1: INT := 1;
	/// Fehler beim Öffnen der Parameterdatei 
	ErrID_2: INT := 2;
	/// ADS - Fehler : Vorgabe Achs ID 
	ErrID_3: INT := 3;
	/// ADS - Fehler : Aktivierung der Parameterliste 
	ErrID_4: INT := 4;
	/// Invalid   CNC Parameter Type 
	ErrID_5: INT := 5;
	/// Invalid   Axis Number  
	ErrID_6: INT := 6;
	/// Invalid   Channel Number  
	ErrID_7: INT := 7;
	/// Invalid   Number  of Parameters 
	ErrID_8: INT := 8;
	/// File Error 
	ErrID_9: INT := 9;
	/// Invalid Channel State 
	ErrID_10: INT := 10;
END_VAR



fbOnTrigger(CLK:= bExecute);

IF fbOnTrigger.Q THEN
	Step 	:= 10;
	nErrorID 	:= 0;
	bError	 := 0;
	bBusy := TRUE;
END_IF

CASE Step OF
0:
	bBusy := FALSE;

10: (* check input parameters *)
	IF (nNumParameters < 1 OR nNumParameters > nMaxParameters) THEN
		nErrorID 	:= ErrID_8;
		Step := 999;
	ELSE
		CASE eParameterType OF
				
			CNC_AxisParameter:
				IF (nLogAxisId <= 0  OR nLogAxisId > MAX_SYS_LOG_AXIS_INDEX) THEN
					nErrorID 	:= ErrID_6;
					Step := 999;
	
				ELSIF (nLogChannelID <= 0 OR nLogChannelID	 > nLogChannelID	) THEN
					nErrorID 	:= ErrID_7;
					Step := 999;
				ELSE
					Step := 12;
				END_IF

			CNC_ChannelParameter:
				IF (nLogChannelID <= 0 OR nLogChannelID > nLogChannelID) THEN
					nErrorID 	:= ErrID_7;
					Step := 999;
				ELSE
					Step := 12;
				END_IF

			CNC_ToolParameter:
				IF (nLogChannelID <= 0 OR nLogChannelID > nLogChannelID) THEN
					nErrorID 	:= ErrID_7;
					Step := 999;
				ELSE
					Step := 12;
				END_IF
	
			CNC_ClampPosition:
				IF (nLogChannelID <= 0 OR nLogChannelID > nLogChannelID) THEN
					nErrorID 	:= ErrID_7;
					Step := 999;
				ELSE
					Step := 12;
				END_IF
	
